LIN {X 0,Y 274.208,Z 1013.96,A -85,B 0,C 180,E1 12726.209,E2 12726.209} C_VEL
LIN {X 0,Y 266.688,Z 1024.123,A -85,B 0,C 180,E1 12721.914,E2 12721.914} C_VEL
LIN {X 0,Y 259.994,Z 1033.612,A -85,B 0,C 180,E1 12716.988,E2 12716.988} C_VEL
LIN {X 0,Y 254.913,Z 1041.187,A -85,B 0,C 180,E1 12711.878,E2 12711.878} C_VEL
LIN {X 0,Y 251.523,Z 1047.053,A -85,B 0,C 180,E1 12706.87,E2 12706.87} C_VEL
LIN {X 0,Y 249.285,Z 1051.783,A -85,B 0,C 180,E1 12701.335,E2 12701.335} C_VEL
LIN {X 0,Y 248.38,Z 1054.512,A -85,B 0,C 180,E1 12696.704,E2 12696.704} C_VEL
LIN {X 0,Y 248.075,Z 1056.133,A -85,B 0,C 180,E1 12692.31,E2 12692.31} C_VEL
LIN {X 0,Y 248.004,Z 1056.84,A -85,B 0,C 180,E1 12687.689,E2 12687.689} C_VEL
LIN {X 0,Y 248.137,Z 1056.355,A -85,B 0,C 180,E1 12682.591,E2 12682.591} C_VEL
LIN {X 0,Y 248.642,Z 1054.659,A -85,B 0,C 180,E1 12677.694,E2 12677.694} C_VEL
LIN {X 0,Y 249.87,Z 1051.971,A -85,B 0,C 180,E1 12673.015,E2 12673.015} C_VEL
LIN {X 0,Y 252.833,Z 1046.979,A -85,B 0,C 180,E1 12667.141,E2 12667.141} C_VEL
LIN {X 0,Y 256.876,Z 1041.112,A -85,B 0,C 180,E1 12662.154,E2 12662.154} C_VEL
LIN {X 0,Y 263.072,Z 1033.015,A -85,B 0,C 180,E1 12656.817,E2 12656.817} C_VEL
LIN {X 0,Y 270.365,Z 1023.771,A -85,B 0,C 180,E1 12652.127,E2 12652.127} C_VEL
LIN {X 0,Y 279.2,Z 1012.904,A -85,B 0,C 180,E1 12647.679,E2 12647.679} C_VEL
LIN {X 0,Y 288.948,Z 1000.521,A -85,B 0,C 180,E1 12643.678,E2 12643.678} C_VEL
LIN {X 0,Y 299.389,Z 987.042,A -85,B 0,C 180,E1 12640.11,E2 12640.11} C_VEL
LIN {X 0,Y 310.24,Z 972.088,A -85,B 0,C 180,E1 12636.937,E2 12636.937} C_VEL
LIN {X 0,Y 320.673,Z 956.975,A -85,B 0,C 180,E1 12634.28,E2 12634.28} C_VEL
LIN {X 0,Y 332.382,Z 938.579,A -85,B 0,C 180,E1 12631.643,E2 12631.643} C_VEL
LIN {X 0,Y 341.93,Z 922.312,A -85,B 0,C 180,E1 12629.715,E2 12629.715} C_VEL
LIN {X 0,Y 353.262,Z 901.024,A -85,B 0,C 180,E1 12627.634,E2 12627.634} C_VEL
LIN {X 0,Y 362.036,Z 882.572,A -85,B 0,C 180,E1 12626.155,E2 12626.155} C_VEL
LIN {X 0,Y 371.461,Z 860.323,A -85,B 0,C 180,E1 12624.686,E2 12624.686} C_VEL
LIN {X 0,Y 379.053,Z 839.359,A -85,B 0,C 180,E1 12623.558,E2 12623.558} C_VEL
LIN {X 0,Y 386.253,Z 816.382,A -85,B 0,C 180,E1 12622.555,E2 12622.555} C_VEL
LIN {X 0,Y 392.125,Z 792.972,A -85,B 0,C 180,E1 12621.762,E2 12621.762} C_VEL
LIN {X 0,Y 396.905,Z 769.324,A -85,B 0,C 180,E1 12621.142,E2 12621.142} C_VEL
LIN {X 0,Y 400.292,Z 744.689,A -85,B 0,C 180,E1 12620.665,E2 12620.665} C_VEL
LIN {X 0,Y 415.264,Z 580.278,A -85,B 0,C 180,E1 12618.096,E2 12618.096} C_VEL
LIN {X 0,Y 415.202,Z 577.101,A -85,B 0,C 180,E1 12617.904,E2 12617.904} C_VEL
LIN {X 0,Y 414.493,Z 574.251,A -85,B 0,C 180,E1 12617.461,E2 12617.461} C_VEL
LIN {X 0,Y 412.986,Z 571.866,A -85,B 0,C 180,E1 12616.684,E2 12616.684} C_VEL
LIN {X 0,Y 410.26,Z 568.824,A -85,B 0,C 180,E1 12615.251,E2 12615.251} C_VEL
LIN {X 0,Y 405.888,Z 561,A -85,B 0,C 180,E1 12612.376,E2 12612.376} C_VEL
LIN {X 0,Y 403.184,Z 556.35,A -85,B 0,C 180,E1 12610.214,E2 12610.214} C_VEL
LIN {X 0,Y 401.232,Z 552.898,A -85,B 0,C 180,E1 12608.311,E2 12608.311} C_VEL
LIN {X 0,Y 399.029,Z 548.877,A -85,B 0,C 180,E1 12605.464,E2 12605.464} C_VEL
LIN {X 0,Y 397.148,Z 544.545,A -85,B 0,C 180,E1 12599.134,E2 12599.134} C_VEL
LIN {X 0,Y 399.305,Z 549.372,A -85,B 0,C 180,E1 12592.446,E2 12592.446} C_VEL
LIN {X 0,Y 402.053,Z 554.34,A -85,B 0,C 180,E1 12589.178,E2 12589.178} C_VEL
LIN {X 0,Y 404.963,Z 559.417,A -85,B 0,C 180,E1 12586.652,E2 12586.652} C_VEL
LIN {X 0,Y 408.355,Z 565.354,A -85,B 0,C 180,E1 12584.265,E2 12584.265} C_VEL
LIN {X 0,Y 413.221,Z 576.035,A -85,B 0,C 180,E1 12581.314,E2 12581.314} C_VEL
LIN {X 0,Y 396.472,Z 755.864,A -85,B 0,C 180,E1 12578.511,E2 12578.511} C_VEL
LIN {X 0,Y 392.307,Z 782.562,A -85,B 0,C 180,E1 12577.987,E2 12577.987} C_VEL
LIN {X 0,Y 387.69,Z 803.875,A -85,B 0,C 180,E1 12577.456,E2 12577.456} C_VEL
LIN {X 0,Y 381.104,Z 828.129,A -85,B 0,C 180,E1 12576.676,E2 12576.676} C_VEL
LIN {X 0,Y 374.28,Z 848.813,A -85,B 0,C 180,E1 12575.828,E2 12575.828} C_VEL
LIN {X 0,Y 365.745,Z 871.344,A -85,B 0,C 180,E1 12574.679,E2 12574.679} C_VEL
LIN {X 0,Y 356.44,Z 892.358,A -85,B 0,C 180,E1 12573.331,E2 12573.331} C_VEL
LIN {X 0,Y 346.382,Z 912.781,A -85,B 0,C 180,E1 12571.744,E2 12571.744} C_VEL
LIN {X 0,Y 335.391,Z 932.564,A -85,B 0,C 180,E1 12569.833,E2 12569.833} C_VEL
LIN {X 0,Y 324.92,Z 949.901,A -85,B 0,C 180,E1 12567.808,E2 12567.808} C_VEL
LIN {X 0,Y 312.929,Z 968.085,A -85,B 0,C 180,E1 12565.203,E2 12565.203} C_VEL
LIN {X 0,Y 302.254,Z 983.196,A -85,B 0,C 180,E1 12562.556,E2 12562.556} C_VEL
LIN {X 0,Y 290.029,Z 999.531,A -85,B 0,C 180,E1 12559.027,E2 12559.027} C_VEL
LIN {X 0,Y 279.971,Z 1012.354,A -85,B 0,C 180,E1 12555.584,E2 12555.584} C_VEL
LIN {X 0,Y 269.185,Z 1025.802,A -85,B 0,C 180,E1 12551.107,E2 12551.107} C_VEL
LIN {X 0,Y 260.773,Z 1036.213,A -85,B 0,C 180,E1 12546.738,E2 12546.738} C_VEL
LIN {X 0,Y 252.94,Z 1046.262,A -85,B 0,C 180,E1 12541.454,E2 12541.454} C_VEL
LIN {X 0,Y 247.478,Z 1053.723,A -85,B 0,C 180,E1 12536.387,E2 12536.387} C_VEL
LIN {X 0,Y 243.363,Z 1060.291,A -85,B 0,C 180,E1 12530.692,E2 12530.692} C_VEL
LIN {X 0,Y 241.068,Z 1064.832,A -85,B 0,C 180,E1 12525.148,E2 12525.148} C_VEL
LIN {X 0,Y 240.171,Z 1067.628,A -85,B 0,C 180,E1 12520.313,E2 12520.313} C_VEL
LIN {X 0,Y 239.975,Z 1069.472,A -85,B 0,C 180,E1 12515.02,E2 12515.02} C_VEL
LIN {X 0,Y 240.024,Z 1069.836,A -85,B 0,C 180,E1 12510,E2 12510} C_VEL
LIN {X 0,Y 239.982,Z 1069.112,A -85,B 0,C 180,E1 12505.46,E2 12505.46} C_VEL
LIN {X 0,Y 240.062,Z 1067.493,A -85,B 0,C 180,E1 12501.135,E2 12501.135} C_VEL
LIN {X 0,Y 240.688,Z 1064.623,A -85,B 0,C 180,E1 12496.303,E2 12496.303} C_VEL
LIN {X 0,Y 242.774,Z 1059.401,A -85,B 0,C 180,E1 12490.262,E2 12490.262} C_VEL
LIN {X 0,Y 245.938,Z 1053.504,A -85,B 0,C 180,E1 12485.244,E2 12485.244} C_VEL
LIN {X 0,Y 251.056,Z 1045.569,A -85,B 0,C 180,E1 12479.879,E2 12479.879} C_VEL
LIN {X 0,Y 257.954,Z 1035.663,A -85,B 0,C 180,E1 12474.721,E2 12474.721} C_VEL
LIN {X 0,Y 266.254,Z 1024.474,A -85,B 0,C 180,E1 12470.006,E2 12470.006} C_VEL
LIN {X 0,Y 275.494,Z 1011.927,A -85,B 0,C 180,E1 12465.825,E2 12465.825} C_VEL
LIN {X 0,Y 285.04,Z 998.91,A -85,B 0,C 180,E1 12462.255,E2 12462.255} C_VEL
LIN {X 0,Y 296.15,Z 983.09,A -85,B 0,C 180,E1 12458.747,E2 12458.747} C_VEL
LIN {X 0,Y 306.358,Z 967.847,A -85,B 0,C 180,E1 12455.979,E2 12455.979} C_VEL
LIN {X 0,Y 317.965,Z 949.305,A -85,B 0,C 180,E1 12453.23,E2 12453.23} C_VEL
LIN {X 0,Y 327.782,Z 932.315,A -85,B 0,C 180,E1 12451.168,E2 12451.168} C_VEL
LIN {X 0,Y 338.722,Z 911.666,A -85,B 0,C 180,E1 12449.1,E2 12449.1} C_VEL
LIN {X 0,Y 347.872,Z 892.386,A -85,B 0,C 180,E1 12447.536,E2 12447.536} C_VEL
LIN {X 0,Y 357.142,Z 870.654,A -85,B 0,C 180,E1 12446.076,E2 12446.076} C_VEL
LIN {X 0,Y 364.973,Z 849.253,A -85,B 0,C 180,E1 12444.931,E2 12444.931} C_VEL
LIN {X 0,Y 371.657,Z 828.377,A -85,B 0,C 180,E1 12444.024,E2 12444.024} C_VEL
LIN {X 0,Y 378.109,Z 803.884,A -85,B 0,C 180,E1 12443.192,E2 12443.192} C_VEL
LIN {X 0,Y 382.633,Z 782.361,A -85,B 0,C 180,E1 12442.628,E2 12442.628} C_VEL
LIN {X 0,Y 386.671,Z 755.374,A -85,B 0,C 180,E1 12442.077,E2 12442.077} C_VEL
LIN {X 0,Y 403.402,Z 568.894,A -85,B 0,C 180,E1 12439.098,E2 12439.098} C_VEL
LIN {X 0,Y 398.244,Z 557.633,A -85,B 0,C 180,E1 12436.332,E2 12436.332} C_VEL
LIN {X 0,Y 393.971,Z 550.114,A -85,B 0,C 180,E1 12433.727,E2 12433.727} C_VEL
LIN {X 0,Y 390.379,Z 543.824,A -85,B 0,C 180,E1 12431.075,E2 12431.075} C_VEL
LIN {X 0,Y 387.521,Z 539.169,A -85,B 0,C 180,E1 12428.457,E2 12428.457} C_VEL
LIN {X 0,Y 385.179,Z 535.036,A -85,B 0,C 180,E1 12425.512,E2 12425.512} C_VEL
LIN {X 0,Y 383.121,Z 530.299,A -85,B 0,C 180,E1 12418.654,E2 12418.654} C_VEL
LIN {X 0,Y 385.47,Z 535.482,A -85,B 0,C 180,E1 12411.648,E2 12411.648} C_VEL
LIN {X 0,Y 388.46,Z 540.683,A -85,B 0,C 180,E1 12408.192,E2 12408.192} C_VEL
LIN {X 0,Y 391.35,Z 545.617,A -85,B 0,C 180,E1 12405.726,E2 12405.726} C_VEL
LIN {X 0,Y 395.237,Z 552.118,A -85,B 0,C 180,E1 12403.048,E2 12403.048} C_VEL
LIN {X 0,Y 400.428,Z 561.515,A -85,B 0,C 180,E1 12400.071,E2 12400.071} C_VEL
LIN {X 0,Y 403.438,Z 567.456,A -85,B 0,C 180,E1 12398.544,E2 12398.544} C_VEL
LIN {X 0,Y 387.142,Z 748.135,A -85,B 0,C 180,E1 12395.669,E2 12395.669} C_VEL
LIN {X 0,Y 383.184,Z 774.56,A -85,B 0,C 180,E1 12395.108,E2 12395.108} C_VEL
LIN {X 0,Y 378.931,Z 795.289,A -85,B 0,C 180,E1 12394.524,E2 12394.524} C_VEL
LIN {X 0,Y 372.699,Z 819.594,A -85,B 0,C 180,E1 12393.646,E2 12393.646} C_VEL
LIN {X 0,Y 366.228,Z 840.253,A -85,B 0,C 180,E1 12392.698,E2 12392.698} C_VEL
LIN {X 0,Y 358.451,Z 861.898,A -85,B 0,C 180,E1 12391.484,E2 12391.484} C_VEL
LIN {X 0,Y 349.307,Z 883.51,A -85,B 0,C 180,E1 12389.986,E2 12389.986} C_VEL
LIN {X 0,Y 340.037,Z 903.213,A -85,B 0,C 180,E1 12388.33,E2 12388.33} C_VEL
LIN {X 0,Y 329.424,Z 923.215,A -85,B 0,C 180,E1 12386.27,E2 12386.27} C_VEL
LIN {X 0,Y 319.951,Z 939.603,A -85,B 0,C 180,E1 12384.239,E2 12384.239} C_VEL
LIN {X 0,Y 308.213,Z 958.246,A -85,B 0,C 180,E1 12381.429,E2 12381.429} C_VEL
LIN {X 0,Y 298.169,Z 973.091,A -85,B 0,C 180,E1 12378.692,E2 12378.692} C_VEL
LIN {X 0,Y 286.701,Z 989.113,A -85,B 0,C 180,E1 12375.07,E2 12375.07} C_VEL
LIN {X 0,Y 277.303,Z 1001.648,A -85,B 0,C 180,E1 12371.564,E2 12371.564} C_VEL
LIN {X 0,Y 267.668,Z 1014.257,A -85,B 0,C 180,E1 12367.24,E2 12367.24} C_VEL
LIN {X 0,Y 259.797,Z 1024.412,A -85,B 0,C 180,E1 12362.866,E2 12362.866} C_VEL
LIN {X 0,Y 252.758,Z 1033.885,A -85,B 0,C 180,E1 12357.827,E2 12357.827} C_VEL
LIN {X 0,Y 247.387,Z 1041.451,A -85,B 0,C 180,E1 12352.58,E2 12352.58} C_VEL
LIN {X 0,Y 243.652,Z 1047.556,A -85,B 0,C 180,E1 12347.186,E2 12347.186} C_VEL
LIN {X 0,Y 241.317,Z 1052.178,A -85,B 0,C 180,E1 12341.472,E2 12341.472} C_VEL
LIN {X 0,Y 240.381,Z 1054.854,A -85,B 0,C 180,E1 12336.688,E2 12336.688} C_VEL
LIN {X 0,Y 240.066,Z 1056.49,A -85,B 0,C 180,E1 12331.909,E2 12331.909} C_VEL
LIN {X 0,Y 240.014,Z 1057.097,A -85,B 0,C 180,E1 12326.895,E2 12326.895} C_VEL
LIN {X 0,Y 240.171,Z 1056.429,A -85,B 0,C 180,E1 12321.862,E2 12321.862} C_VEL
LIN {X 0,Y 240.764,Z 1054.748,A -85,B 0,C 180,E1 12317.041,E2 12317.041} C_VEL
LIN {X 0,Y 242.354,Z 1051.699,A -85,B 0,C 180,E1 12311.726,E2 12311.726} C_VEL
LIN {X 0,Y 245.555,Z 1046.718,A -85,B 0,C 180,E1 12305.971,E2 12305.971} C_VEL
LIN {X 0,Y 249.825,Z 1040.987,A -85,B 0,C 180,E1 12301.034,E2 12301.034} C_VEL
LIN {X 0,Y 256.801,Z 1032.373,A -85,B 0,C 180,E1 12295.356,E2 12295.356} C_VEL
LIN {X 0,Y 264.258,Z 1023.467,A -85,B 0,C 180,E1 12290.81,E2 12290.81} C_VEL
LIN {X 0,Y 274.029,Z 1011.899,A -85,B 0,C 180,E1 12286.11,E2 12286.11} C_VEL
LIN {X 0,Y 283.806,Z 1000.013,A -85,B 0,C 180,E1 12282.281,E2 12282.281} C_VEL
LIN {X 0,Y 295.269,Z 985.638,A -85,B 0,C 180,E1 12278.533,E2 12278.533} C_VEL
LIN {X 0,Y 305.967,Z 971.336,A -85,B 0,C 180,E1 12275.539,E2 12275.539} C_VEL
LIN {X 0,Y 317.421,Z 955.203,A -85,B 0,C 180,E1 12272.748,E2 12272.748} C_VEL
LIN {X 0,Y 328.836,Z 937.519,A -85,B 0,C 180,E1 12270.281,E2 12270.281} C_VEL
LIN {X 0,Y 339.38,Z 919.914,A -85,B 0,C 180,E1 12268.246,E2 12268.246} C_VEL
LIN {X 0,Y 350.287,Z 899.549,A -85,B 0,C 180,E1 12266.323,E2 12266.323} C_VEL
LIN {X 0,Y 358.905,Z 881.731,A -85,B 0,C 180,E1 12264.93,E2 12264.93} C_VEL
LIN {X 0,Y 368.941,Z 858.156,A -85,B 0,C 180,E1 12263.42,E2 12263.42} C_VEL
LIN {X 0,Y 376.287,Z 838.102,A -85,B 0,C 180,E1 12262.373,E2 12262.373} C_VEL
LIN {X 0,Y 383.819,Z 813.925,A -85,B 0,C 180,E1 12261.358,E2 12261.358} C_VEL
LIN {X 0,Y 389.378,Z 791.903,A -85,B 0,C 180,E1 12260.635,E2 12260.635} C_VEL
LIN {X 0,Y 394.305,Z 767.229,A -85,B 0,C 180,E1 12260.014,E2 12260.014} C_VEL
LIN {X 0,Y 397.509,Z 743.917,A -85,B 0,C 180,E1 12259.577,E2 12259.577} C_VEL
LIN {X 0,Y 413.233,Z 574.497,A -85,B 0,C 180,E1 12256.939,E2 12256.939} C_VEL
LIN {X 0,Y 410.26,Z 568.824,A -85,B 0,C 180,E1 12255.251,E2 12255.251} C_VEL
LIN {X 0,Y 408.323,Z 566.877,A -85,B 0,C 180,E1 12254.153,E2 12254.153} C_VEL
LIN {X 0,Y 402.936,Z 565.423,A -85,B 0,C 180,E1 12250.841,E2 12250.841} C_VEL
LIN {X 0,Y 402.359,Z 564.773,A -85,B 0,C 180,E1 12250.379,E2 12250.379} C_VEL
LIN {X 0,Y 399.981,Z 560.605,A -85,B 0,C 180,E1 12248.047,E2 12248.047} C_VEL
LIN {X 0,Y 397.86,Z 556.677,A -85,B 0,C 180,E1 12245.191,E2 12245.191} C_VEL
LIN {X 0,Y 396.169,Z 552.519,A -85,B 0,C 180,E1 12239.132,E2 12239.132} C_VEL
LIN {X 0,Y 398.223,Z 557.306,A -85,B 0,C 180,E1 12232.57,E2 12232.57} C_VEL
LIN {X 0,Y 400.781,Z 562.036,A -85,B 0,C 180,E1 12229.434,E2 12229.434} C_VEL
LIN {X 0,Y 403.525,Z 566.964,A -85,B 0,C 180,E1 12226.968,E2 12226.968} C_VEL
LIN {X 0,Y 406.77,Z 572.828,A -85,B 0,C 180,E1 12224.605,E2 12224.605} C_VEL
LIN {X 0,Y 410.341,Z 581.211,A -85,B 0,C 180,E1 12222.297,E2 12222.297} C_VEL
LIN {X 0,Y 393.726,Z 755.676,A -85,B 0,C 180,E1 12219.606,E2 12219.606} C_VEL
LIN {X 0,Y 389.508,Z 782.287,A -85,B 0,C 180,E1 12219.091,E2 12219.091} C_VEL
LIN {X 0,Y 384.811,Z 803.636,A -85,B 0,C 180,E1 12218.571,E2 12218.571} C_VEL
LIN {X 0,Y 377.998,Z 828.265,A -85,B 0,C 180,E1 12217.794,E2 12217.794} C_VEL
LIN {X 0,Y 371.058,Z 848.906,A -85,B 0,C 180,E1 12216.961,E2 12216.961} C_VEL
LIN {X 0,Y 362.252,Z 871.633,A -85,B 0,C 180,E1 12215.818,E2 12215.818} C_VEL
LIN {X 0,Y 352.801,Z 892.535,A -85,B 0,C 180,E1 12214.493,E2 12214.493} C_VEL
LIN {X 0,Y 342.316,Z 913.337,A -85,B 0,C 180,E1 12212.892,E2 12212.892} C_VEL
LIN {X 0,Y 331.006,Z 933.122,A -85,B 0,C 180,E1 12210.987,E2 12210.987} C_VEL
LIN {X 0,Y 319.94,Z 950.948,A -85,B 0,C 180,E1 12208.905,E2 12208.905} C_VEL
LIN {X 0,Y 307.654,Z 968.923,A -85,B 0,C 180,E1 12206.306,E2 12206.306} C_VEL
LIN {X 0,Y 296.416,Z 984.325,A -85,B 0,C 180,E1 12203.58,E2 12203.58} C_VEL
LIN {X 0,Y 284.108,Z 1000.112,A -85,B 0,C 180,E1 12200.106,E2 12200.106} C_VEL
LIN {X 0,Y 274.242,Z 1012.221,A -85,B 0,C 180,E1 12196.82,E2 12196.82} C_VEL
LIN {X 0,Y 262.999,Z 1025.652,A -85,B 0,C 180,E1 12192.294,E2 12192.294} C_VEL
LIN {X 0,Y 254.566,Z 1035.589,A -85,B 0,C 180,E1 12188.073,E2 12188.073} C_VEL
LIN {X 0,Y 246.508,Z 1045.405,A -85,B 0,C 180,E1 12182.898,E2 12182.898} C_VEL
LIN {X 0,Y 240.341,Z 1053.235,A -85,B 0,C 180,E1 12177.503,E2 12177.503} C_VEL
LIN {X 0,Y 235.845,Z 1059.872,A -85,B 0,C 180,E1 12171.645,E2 12171.645} C_VEL
LIN {X 0,Y 233.202,Z 1064.635,A -85,B 0,C 180,E1 12165.672,E2 12165.672} C_VEL
LIN {X 0,Y 232.206,Z 1067.427,A -85,B 0,C 180,E1 12160.67,E2 12160.67} C_VEL
LIN {X 0,Y 231.976,Z 1069.266,A -85,B 0,C 180,E1 12155.193,E2 12155.193} C_VEL
LIN {X 0,Y 232.019,Z 1069.641,A -85,B 0,C 180,E1 12150.247,E2 12150.247} C_VEL
LIN {X 0,Y 231.984,Z 1068.958,A -85,B 0,C 180,E1 12145.55,E2 12145.55} C_VEL
LIN {X 0,Y 232.065,Z 1067.379,A -85,B 0,C 180,E1 12141.077,E2 12141.077} C_VEL
LIN {X 0,Y 232.701,Z 1064.624,A -85,B 0,C 180,E1 12136.192,E2 12136.192} C_VEL
LIN {X 0,Y 234.7,Z 1059.909,A -85,B 0,C 180,E1 12130.31,E2 12130.31} C_VEL
LIN {X 0,Y 238.268,Z 1053.553,A -85,B 0,C 180,E1 12124.657,E2 12124.657} C_VEL
LIN {X 0,Y 243.373,Z 1046.025,A -85,B 0,C 180,E1 12119.373,E2 12119.373} C_VEL
LIN {X 0,Y 250.514,Z 1036.315,A -85,B 0,C 180,E1 12114.075,E2 12114.075} C_VEL
LIN {X 0,Y 258.183,Z 1026.358,A -85,B 0,C 180,E1 12109.703,E2 12109.703} C_VEL
LIN {X 0,Y 268.617,Z 1012.911,A -85,B 0,C 180,E1 12104.989,E2 12104.989} C_VEL
LIN {X 0,Y 277.893,Z 1000.729,A -85,B 0,C 180,E1 12101.547,E2 12101.547} C_VEL
LIN {X 0,Y 289.353,Z 985.184,A -85,B 0,C 180,E1 12097.959,E2 12097.959} C_VEL
LIN {X 0,Y 299.7,Z 970.261,A -85,B 0,C 180,E1 12095.175,E2 12095.175} C_VEL
LIN {X 0,Y 311.165,Z 952.835,A -85,B 0,C 180,E1 12092.487,E2 12092.487} C_VEL
LIN {X 0,Y 322.546,Z 933.775,A -85,B 0,C 180,E1 12090.129,E2 12090.129} C_VEL
LIN {X 0,Y 333.349,Z 914.165,A -85,B 0,C 180,E1 12088.132,E2 12088.132} C_VEL
LIN {X 0,Y 343.386,Z 893.65,A -85,B 0,C 180,E1 12086.456,E2 12086.456} C_VEL
LIN {X 0,Y 352.222,Z 873.559,A -85,B 0,C 180,E1 12085.099,E2 12085.099} C_VEL
LIN {X 0,Y 360.979,Z 850.598,A -85,B 0,C 180,E1 12083.854,E2 12083.854} C_VEL
LIN {X 0,Y 367.441,Z 830.993,A -85,B 0,C 180,E1 12083,E2 12083} C_VEL
LIN {X 0,Y 374.212,Z 806.578,A -85,B 0,C 180,E1 12082.153,E2 12082.153} C_VEL
LIN {X 0,Y 379.062,Z 784.332,A -85,B 0,C 180,E1 12081.567,E2 12081.567} C_VEL
LIN {X 0,Y 383.117,Z 759.514,A -85,B 0,C 180,E1 12081.049,E2 12081.049} C_VEL
LIN {X 0,Y 388.393,Z 704.087,A -85,B 0,C 180,E1 12080.146,E2 12080.146} C_VEL
LIN {X 0,Y 400.252,Z 573.446,A -85,B 0,C 180,E1 12078.083,E2 12078.083} C_VEL
LIN {X 0,Y 395.946,Z 563.972,A -85,B 0,C 180,E1 12075.639,E2 12075.639} C_VEL
LIN {X 0,Y 391.725,Z 556.337,A -85,B 0,C 180,E1 12072.906,E2 12072.906} C_VEL
LIN {X 0,Y 388.594,Z 550.898,A -85,B 0,C 180,E1 12070.452,E2 12070.452} C_VEL
LIN {X 0,Y 386.254,Z 546.876,A -85,B 0,C 180,E1 12068.185,E2 12068.185} C_VEL
LIN {X 0,Y 383.997,Z 542.829,A -85,B 0,C 180,E1 12065.229,E2 12065.229} C_VEL
LIN {X 0,Y 382.142,Z 538.278,A -85,B 0,C 180,E1 12058.651,E2 12058.651} C_VEL
LIN {X 0,Y 384.382,Z 543.419,A -85,B 0,C 180,E1 12051.774,E2 12051.774} C_VEL
LIN {X 0,Y 387.171,Z 548.383,A -85,B 0,C 180,E1 12048.454,E2 12048.454} C_VEL
LIN {X 0,Y 389.894,Z 553.166,A -85,B 0,C 180,E1 12046.051,E2 12046.051} C_VEL
LIN {X 0,Y 393.621,Z 559.599,A -85,B 0,C 180,E1 12043.395,E2 12043.395} C_VEL
LIN {X 0,Y 398.687,Z 569.021,A -85,B 0,C 180,E1 12040.401,E2 12040.401} C_VEL
LIN {X 0,Y 400.284,Z 572.367,A -85,B 0,C 180,E1 12039.544,E2 12039.544} C_VEL
LIN {X 0,Y 384.057,Z 748.302,A -85,B 0,C 180,E1 12036.767,E2 12036.767} C_VEL
LIN {X 0,Y 380.026,Z 774.745,A -85,B 0,C 180,E1 12036.213,E2 12036.213} C_VEL
LIN {X 0,Y 375.691,Z 795.491,A -85,B 0,C 180,E1 12035.638,E2 12035.638} C_VEL
LIN {X 0,Y 369.224,Z 820.189,A -85,B 0,C 180,E1 12034.756,E2 12034.756} C_VEL
LIN {X 0,Y 362.643,Z 840.766,A -85,B 0,C 180,E1 12033.822,E2 12033.822} C_VEL
LIN {X 0,Y 354.698,Z 862.408,A -85,B 0,C 180,E1 12032.621,E2 12032.621} C_VEL
LIN {X 0,Y 345.362,Z 883.966,A -85,B 0,C 180,E1 12031.139,E2 12031.139} C_VEL
LIN {X 0,Y 335.768,Z 903.879,A -85,B 0,C 180,E1 12029.477,E2 12029.477} C_VEL
LIN {X 0,Y 325.015,Z 923.613,A -85,B 0,C 180,E1 12027.452,E2 12027.452} C_VEL
LIN {X 0,Y 314.859,Z 940.708,A -85,B 0,C 180,E1 12025.336,E2 12025.336} C_VEL
LIN {X 0,Y 303.227,Z 958.602,A -85,B 0,C 180,E1 12022.627,E2 12022.627} C_VEL
LIN {X 0,Y 292.874,Z 973.436,A -85,B 0,C 180,E1 12019.885,E2 12019.885} C_VEL
LIN {X 0,Y 281.008,Z 989.437,A -85,B 0,C 180,E1 12016.246,E2 12016.246} C_VEL
LIN {X 0,Y 271.257,Z 1001.963,A -85,B 0,C 180,E1 12012.707,E2 12012.707} C_VEL
LIN {X 0,Y 261.14,Z 1014.647,A -85,B 0,C 180,E1 12008.285,E2 12008.285} C_VEL
LIN {X 0,Y 252.983,Z 1024.7,A -85,B 0,C 180,E1 12003.868,E2 12003.868} C_VEL
LIN {X 0,Y 245.579,Z 1034.158,A -85,B 0,C 180,E1 11998.714,E2 11998.714} C_VEL
LIN {X 0,Y 239.901,Z 1041.714,A -85,B 0,C 180,E1 11993.325,E2 11993.325} C_VEL
LIN {X 0,Y 235.924,Z 1047.812,A -85,B 0,C 180,E1 11987.767,E2 11987.767} C_VEL
LIN {X 0,Y 233.421,Z 1052.417,A -85,B 0,C 180,E1 11981.865,E2 11981.865} C_VEL
LIN {X 0,Y 232.411,Z 1055.085,A -85,B 0,C 180,E1 11976.919,E2 11976.919} C_VEL
LIN {X 0,Y 232.071,Z 1056.714,A -85,B 0,C 180,E1 11971.975,E2 11971.975} C_VEL
LIN {X 0,Y 232.018,Z 1057.307,A -85,B 0,C 180,E1 11966.788,E2 11966.788} C_VEL
LIN {X 0,Y 232.196,Z 1056.634,A -85,B 0,C 180,E1 11961.581,E2 11961.581} C_VEL
LIN {X 0,Y 232.853,Z 1054.948,A -85,B 0,C 180,E1 11956.592,E2 11956.592} C_VEL
LIN {X 0,Y 234.592,Z 1051.893,A -85,B 0,C 180,E1 11951.099,E2 11951.099} C_VEL
LIN {X 0,Y 238.088,Z 1046.847,A -85,B 0,C 180,E1 11945.112,E2 11945.112} C_VEL
LIN {X 0,Y 242.615,Z 1041.161,A -85,B 0,C 180,E1 11940.087,E2 11940.087} C_VEL
LIN {X 0,Y 250.02,Z 1032.531,A -85,B 0,C 180,E1 11934.275,E2 11934.275} C_VEL
LIN {X 0,Y 257.882,Z 1023.616,A -85,B 0,C 180,E1 11929.646,E2 11929.646} C_VEL
LIN {X 0,Y 268.413,Z 1011.672,A -85,B 0,C 180,E1 11924.754,E2 11924.754} C_VEL
LIN {X 0,Y 278.302,Z 1000.135,A -85,B 0,C 180,E1 11921.019,E2 11921.019} C_VEL
LIN {X 0,Y 290.19,Z 985.74,A -85,B 0,C 180,E1 11917.256,E2 11917.256} C_VEL
LIN {X 0,Y 301.246,Z 971.426,A -85,B 0,C 180,E1 11914.261,E2 11914.261} C_VEL
LIN {X 0,Y 313.044,Z 955.275,A -85,B 0,C 180,E1 11911.48,E2 11911.48} C_VEL
LIN {X 0,Y 324.773,Z 937.569,A -85,B 0,C 180,E1 11909.031,E2 11909.031} C_VEL
LIN {X 0,Y 335.952,Z 919.34,A -85,B 0,C 180,E1 11906.951,E2 11906.951} C_VEL
LIN {X 0,Y 346.746,Z 899.544,A -85,B 0,C 180,E1 11905.114,E2 11905.114} C_VEL
LIN {X 0,Y 355.593,Z 881.622,A -85,B 0,C 180,E1 11903.736,E2 11903.736} C_VEL
LIN {X 0,Y 365.537,Z 858.721,A -85,B 0,C 180,E1 11902.29,E2 11902.29} C_VEL
LIN {X 0,Y 372.878,Z 839.111,A -85,B 0,C 180,E1 11901.277,E2 11901.277} C_VEL
LIN {X 0,Y 380.332,Z 815.968,A -85,B 0,C 180,E1 11900.306,E2 11900.306} C_VEL
LIN {X 0,Y 386.25,Z 793.125,A -85,B 0,C 180,E1 11899.56,E2 11899.56} C_VEL
LIN {X 0,Y 391.244,Z 769.089,A -85,B 0,C 180,E1 11898.954,E2 11898.954} C_VEL
LIN {X 0,Y 394.683,Z 744.791,A -85,B 0,C 180,E1 11898.5,E2 11898.5} C_VEL
LIN {X 0,Y 410.348,Z 579.625,A -85,B 0,C 180,E1 11895.946,E2 11895.946} C_VEL
LIN {X 0,Y 405.942,Z 571.377,A -85,B 0,C 180,E1 11893.17,E2 11893.17} C_VEL
LIN {X 0,Y 402.359,Z 564.773,A -85,B 0,C 180,E1 11890.379,E2 11890.379} C_VEL
LIN {X 0,Y 400.956,Z 563.777,A -85,B 0,C 180,E1 11889.221,E2 11889.221} C_VEL
LIN {X 0,Y 397.256,Z 564.937,A -85,B 0,C 180,E1 11885.734,E2 11885.734} C_VEL
LIN {X 0,Y 396.971,Z 564.739,A -85,B 0,C 180,E1 11885.334,E2 11885.334} C_VEL
LIN {X 0,Y 395.189,Z 560.495,A -85,B 0,C 180,E1 11879.13,E2 11879.13} C_VEL
LIN {X 0,Y 397.102,Z 565.119,A -85,B 0,C 180,E1 11872.767,E2 11872.767} C_VEL
LIN {X 0,Y 399.583,Z 569.876,A -85,B 0,C 180,E1 11869.62,E2 11869.62} C_VEL
LIN {X 0,Y 402.269,Z 574.828,A -85,B 0,C 180,E1 11867.146,E2 11867.146} C_VEL
LIN {X 0,Y 405.294,Z 580.545,A -85,B 0,C 180,E1 11864.877,E2 11864.877} C_VEL
LIN {X 0,Y 407.597,Z 586.184,A -85,B 0,C 180,E1 11863.301,E2 11863.301} C_VEL
LIN {X 0,Y 391.12,Z 755.536,A -85,B 0,C 180,E1 11860.715,E2 11860.715} C_VEL
LIN {X 0,Y 386.856,Z 782.013,A -85,B 0,C 180,E1 11860.211,E2 11860.211} C_VEL
LIN {X 0,Y 382.072,Z 803.435,A -85,B 0,C 180,E1 11859.701,E2 11859.701} C_VEL
LIN {X 0,Y 375.038,Z 828.403,A -85,B 0,C 180,E1 11858.929,E2 11858.929} C_VEL
LIN {X 0,Y 367.984,Z 849.001,A -85,B 0,C 180,E1 11858.114,E2 11858.114} C_VEL
LIN {X 0,Y 359.022,Z 871.665,A -85,B 0,C 180,E1 11856.993,E2 11856.993} C_VEL
LIN {X 0,Y 349.433,Z 892.46,A -85,B 0,C 180,E1 11855.696,E2 11855.696} C_VEL
LIN {X 0,Y 338.891,Z 912.953,A -85,B 0,C 180,E1 11854.144,E2 11854.144} C_VEL
LIN {X 0,Y 327.505,Z 932.463,A -85,B 0,C 180,E1 11852.299,E2 11852.299} C_VEL
LIN {X 0,Y 316.516,Z 949.77,A -85,B 0,C 180,E1 11850.313,E2 11850.313} C_VEL
LIN {X 0,Y 303.867,Z 967.902,A -85,B 0,C 180,E1 11847.744,E2 11847.744} C_VEL
LIN {X 0,Y 293.193,Z 982.14,A -85,B 0,C 180,E1 11845.275,E2 11845.275} C_VEL
LIN {X 0,Y 280.683,Z 997.872,A -85,B 0,C 180,E1 11841.932,E2 11841.932} C_VEL
LIN {X 0,Y 269.384,Z 1011.222,A -85,B 0,C 180,E1 11838.363,E2 11838.363} C_VEL
LIN {X 0,Y 258.376,Z 1023.94,A -85,B 0,C 180,E1 11834.153,E2 11834.153} C_VEL
LIN {X 0,Y 248.504,Z 1034.966,A -85,B 0,C 180,E1 11829.474,E2 11829.474} C_VEL
LIN {X 0,Y 239.962,Z 1044.827,A -85,B 0,C 180,E1 11824.231,E2 11824.231} C_VEL
LIN {X 0,Y 233.287,Z 1052.746,A -85,B 0,C 180,E1 11818.688,E2 11818.688} C_VEL
LIN {X 0,Y 228.711,Z 1058.908,A -85,B 0,C 180,E1 11813.17,E2 11813.17} C_VEL
LIN {X 0,Y 225.515,Z 1064.125,A -85,B 0,C 180,E1 11806.723,E2 11806.723} C_VEL
LIN {X 0,Y 224.312,Z 1066.99,A -85,B 0,C 180,E1 11801.572,E2 11801.572} C_VEL
LIN {X 0,Y 223.979,Z 1068.777,A -85,B 0,C 180,E1 11796.408,E2 11796.408} C_VEL
LIN {X 0,Y 224.01,Z 1069.469,A -85,B 0,C 180,E1 11791.279,E2 11791.279} C_VEL
LIN {X 0,Y 223.991,Z 1069.015,A -85,B 0,C 180,E1 11786.417,E2 11786.417} C_VEL
LIN {X 0,Y 224.053,Z 1067.383,A -85,B 0,C 180,E1 11781.273,E2 11781.273} C_VEL
LIN {X 0,Y 224.71,Z 1064.64,A -85,B 0,C 180,E1 11776.097,E2 11776.097} C_VEL
LIN {X 0,Y 226.6,Z 1060.347,A -85,B 0,C 180,E1 11770.406,E2 11770.406} C_VEL
LIN {X 0,Y 230.424,Z 1053.913,A -85,B 0,C 180,E1 11764.282,E2 11764.282} C_VEL
LIN {X 0,Y 235.435,Z 1046.841,A -85,B 0,C 180,E1 11759.077,E2 11759.077} C_VEL
LIN {X 0,Y 243.47,Z 1036.499,A -85,B 0,C 180,E1 11753.159,E2 11753.159} C_VEL
LIN {X 0,Y 251.465,Z 1026.59,A -85,B 0,C 180,E1 11748.696,E2 11748.696} C_VEL
LIN {X 0,Y 262.304,Z 1013.248,A -85,B 0,C 180,E1 11743.908,E2 11743.908} C_VEL
LIN {X 0,Y 272.513,Z 1000.343,A -85,B 0,C 180,E1 11740.224,E2 11740.224} C_VEL
LIN {X 0,Y 284.845,Z 984.13,A -85,B 0,C 180,E1 11736.5,E2 11736.5} C_VEL
LIN {X 0,Y 295.676,Z 968.974,A -85,B 0,C 180,E1 11733.706,E2 11733.706} C_VEL
LIN {X 0,Y 307.858,Z 950.808,A -85,B 0,C 180,E1 11730.969,E2 11730.969} C_VEL
LIN {X 0,Y 318.866,Z 932.772,A -85,B 0,C 180,E1 11728.783,E2 11728.783} C_VEL
LIN {X 0,Y 329.909,Z 913.124,A -85,B 0,C 180,E1 11726.821,E2 11726.821} C_VEL
LIN {X 0,Y 340.246,Z 892.323,A -85,B 0,C 180,E1 11725.16,E2 11725.16} C_VEL
LIN {X 0,Y 349.638,Z 871.278,A -85,B 0,C 180,E1 11723.776,E2 11723.776} C_VEL
LIN {X 0,Y 358.028,Z 849.339,A -85,B 0,C 180,E1 11722.63,E2 11722.63} C_VEL
LIN {X 0,Y 364.543,Z 829.829,A -85,B 0,C 180,E1 11721.805,E2 11721.805} C_VEL
LIN {X 0,Y 371.552,Z 804.574,A -85,B 0,C 180,E1 11720.962,E2 11720.962} C_VEL
LIN {X 0,Y 376.275,Z 783.017,A -85,B 0,C 180,E1 11720.412,E2 11720.412} C_VEL
LIN {X 0,Y 380.395,Z 757.375,A -85,B 0,C 180,E1 11719.894,E2 11719.894} C_VEL
LIN {X 0,Y 387.886,Z 678.764,A -85,B 0,C 180,E1 11718.639,E2 11718.639} C_VEL
LIN {X 0,Y 397.206,Z 578.193,A -85,B 0,C 180,E1 11717.054,E2 11717.054} C_VEL
LIN {X 0,Y 393.989,Z 570.875,A -85,B 0,C 180,E1 11715.116,E2 11715.116} C_VEL
LIN {X 0,Y 389.653,Z 562.753,A -85,B 0,C 180,E1 11712.147,E2 11712.147} C_VEL
LIN {X 0,Y 387.019,Z 558.202,A -85,B 0,C 180,E1 11709.968,E2 11709.968} C_VEL
LIN {X 0,Y 384.996,Z 554.581,A -85,B 0,C 180,E1 11707.912,E2 11707.912} C_VEL
LIN {X 0,Y 382.923,Z 550.71,A -85,B 0,C 180,E1 11705.093,E2 11705.093} C_VEL
LIN {X 0,Y 381.159,Z 546.277,A -85,B 0,C 180,E1 11698.647,E2 11698.647} C_VEL
LIN {X 0,Y 383.252,Z 551.234,A -85,B 0,C 180,E1 11691.976,E2 11691.976} C_VEL
LIN {X 0,Y 385.89,Z 556.083,A -85,B 0,C 180,E1 11688.718,E2 11688.718} C_VEL
LIN {X 0,Y 388.626,Z 561.047,A -85,B 0,C 180,E1 11686.232,E2 11686.232} C_VEL
LIN {X 0,Y 392.071,Z 567.186,A -85,B 0,C 180,E1 11683.708,E2 11683.708} C_VEL
LIN {X 0,Y 397.023,Z 576.643,A -85,B 0,C 180,E1 11680.698,E2 11680.698} C_VEL
LIN {X 0,Y 397.235,Z 577.499,A -85,B 0,C 180,E1 11680.556,E2 11680.556} C_VEL
LIN {X 0,Y 381.103,Z 748.566,A -85,B 0,C 180,E1 11677.881,E2 11677.881} C_VEL
LIN {X 0,Y 377.011,Z 774.925,A -85,B 0,C 180,E1 11677.336,E2 11677.336} C_VEL
LIN {X 0,Y 372.563,Z 795.837,A -85,B 0,C 180,E1 11676.766,E2 11676.766} C_VEL
LIN {X 0,Y 365.89,Z 820.783,A -85,B 0,C 180,E1 11675.887,E2 11675.887} C_VEL
LIN {X 0,Y 359.201,Z 841.277,A -85,B 0,C 180,E1 11674.968,E2 11674.968} C_VEL
LIN {X 0,Y 350.7,Z 863.813,A -85,B 0,C 180,E1 11673.725,E2 11673.725} C_VEL
LIN {X 0,Y 341.559,Z 884.422,A -85,B 0,C 180,E1 11672.319,E2 11672.319} C_VEL
LIN {X 0,Y 331.921,Z 903.982,A -85,B 0,C 180,E1 11670.703,E2 11670.703} C_VEL
LIN {X 0,Y 320.748,Z 924.011,A -85,B 0,C 180,E1 11668.667,E2 11668.667} C_VEL
LIN {X 0,Y 310.371,Z 941.03,A -85,B 0,C 180,E1 11666.571,E2 11666.571} C_VEL
LIN {X 0,Y 298.317,Z 959.043,A -85,B 0,C 180,E1 11663.849,E2 11663.849} C_VEL
LIN {X 0,Y 287.709,Z 973.781,A -85,B 0,C 180,E1 11661.121,E2 11661.121} C_VEL
LIN {X 0,Y 275.441,Z 989.761,A -85,B 0,C 180,E1 11657.47,E2 11657.47} C_VEL
LIN {X 0,Y 265.709,Z 1001.804,A -85,B 0,C 180,E1 11654.048,E2 11654.048} C_VEL
LIN {X 0,Y 255.317,Z 1014.345,A -85,B 0,C 180,E1 11649.669,E2 11649.669} C_VEL
LIN {X 0,Y 246.25,Z 1024.988,A -85,B 0,C 180,E1 11644.926,E2 11644.926} C_VEL
LIN {X 0,Y 238.464,Z 1034.429,A -85,B 0,C 180,E1 11639.655,E2 11639.655} C_VEL
LIN {X 0,Y 232.457,Z 1041.978,A -85,B 0,C 180,E1 11634.119,E2 11634.119} C_VEL
LIN {X 0,Y 228.221,Z 1048.067,A -85,B 0,C 180,E1 11628.388,E2 11628.388} C_VEL
LIN {X 0,Y 225.534,Z 1052.657,A -85,B 0,C 180,E1 11622.287,E2 11622.287} C_VEL
LIN {X 0,Y 224.445,Z 1055.317,A -85,B 0,C 180,E1 11617.166,E2 11617.166} C_VEL
LIN {X 0,Y 224.076,Z 1056.938,A -85,B 0,C 180,E1 11612.046,E2 11612.046} C_VEL
LIN {X 0,Y 224.022,Z 1057.518,A -85,B 0,C 180,E1 11606.674,E2 11606.674} C_VEL
LIN {X 0,Y 224.227,Z 1056.838,A -85,B 0,C 180,E1 11601.279,E2 11601.279} C_VEL
LIN {X 0,Y 224.953,Z 1055.147,A -85,B 0,C 180,E1 11596.112,E2 11596.112} C_VEL
LIN {X 0,Y 226.857,Z 1052.087,A -85,B 0,C 180,E1 11590.429,E2 11590.429} C_VEL
LIN {X 0,Y 230.594,Z 1047.079,A -85,B 0,C 180,E1 11584.303,E2 11584.303} C_VEL
LIN {X 0,Y 235.517,Z 1041.292,A -85,B 0,C 180,E1 11579.048,E2 11579.048} C_VEL
LIN {X 0,Y 243.335,Z 1032.69,A -85,B 0,C 180,E1 11573.135,E2 11573.135} C_VEL
LIN {X 0,Y 251.188,Z 1024.22,A -85,B 0,C 180,E1 11568.64,E2 11568.64} C_VEL
LIN {X 0,Y 261.331,Z 1013.301,A -85,B 0,C 180,E1 11564.002,E2 11564.002} C_VEL
LIN {X 0,Y 271.895,Z 1001.438,A -85,B 0,C 180,E1 11560.058,E2 11560.058} C_VEL
LIN {X 0,Y 283.435,Z 988.076,A -85,B 0,C 180,E1 11556.455,E2 11556.455} C_VEL
LIN {X 0,Y 295.45,Z 973.104,A -85,B 0,C 180,E1 11553.248,E2 11553.248} C_VEL
LIN {X 0,Y 306.754,Z 958.132,A -85,B 0,C 180,E1 11550.624,E2 11550.624} C_VEL
LIN {X 0,Y 319.664,Z 939.475,A -85,B 0,C 180,E1 11547.982,E2 11547.982} C_VEL
LIN {X 0,Y 329.702,Z 923.628,A -85,B 0,C 180,E1 11546.145,E2 11546.145} C_VEL
LIN {X 0,Y 341.262,Z 903.562,A -85,B 0,C 180,E1 11544.217,E2 11544.217} C_VEL
LIN {X 0,Y 350.777,Z 884.924,A -85,B 0,C 180,E1 11542.759,E2 11542.759} C_VEL
LIN {X 0,Y 360.324,Z 864.084,A -85,B 0,C 180,E1 11541.408,E2 11541.408} C_VEL
LIN {X 0,Y 369.07,Z 841.614,A -85,B 0,C 180,E1 11540.23,E2 11540.23} C_VEL
LIN {X 0,Y 376.17,Z 820.468,A -85,B 0,C 180,E1 11539.332,E2 11539.332} C_VEL
LIN {X 0,Y 382.899,Z 795.872,A -85,B 0,C 180,E1 11538.513,E2 11538.513} C_VEL
LIN {X 0,Y 387.518,Z 774.707,A -85,B 0,C 180,E1 11537.969,E2 11537.969} C_VEL
LIN {X 0,Y 391.73,Z 747.973,A -85,B 0,C 180,E1 11537.447,E2 11537.447} C_VEL
LIN {X 0,Y 407.604,Z 585.037,A -85,B 0,C 180,E1 11534.965,E2 11534.965} C_VEL
LIN {X 0,Y 403.504,Z 577.084,A -85,B 0,C 180,E1 11532.159,E2 11532.159} C_VEL
LIN {X 0,Y 400.575,Z 571.719,A -85,B 0,C 180,E1 11529.7,E2 11529.7} C_VEL
LIN {X 0,Y 398.739,Z 568.31,A -85,B 0,C 180,E1 11527.783,E2 11527.783} C_VEL
LIN {X 0,Y 396.971,Z 564.739,A -85,B 0,C 180,E1 11525.334,E2 11525.334} C_VEL
LIN {X 0,Y 396.187,Z 564.939,A -85,B 0,C 180,E1 11524.219,E2 11524.219} C_VEL
LIN {X 0,Y 394.357,Z 569.171,A -85,B 0,C 180,E1 11521.132,E2 11521.132} C_VEL
LIN {X 0,Y 394.191,Z 569.196,A -85,B 0,C 180,E1 11520.245,E2 11520.245} C_VEL
LIN {X 0,Y 394.201,Z 568.561,A -85,B 0,C 180,E1 11518.983,E2 11518.983} C_VEL
LIN {X 0,Y 395.985,Z 572.93,A -85,B 0,C 180,E1 11512.966,E2 11512.966} C_VEL
LIN {X 0,Y 398.325,Z 577.571,A -85,B 0,C 180,E1 11509.88,E2 11509.88} C_VEL
LIN {X 0,Y 400.85,Z 582.375,A -85,B 0,C 180,E1 11507.466,E2 11507.466} C_VEL
LIN {X 0,Y 403.733,Z 588.041,A -85,B 0,C 180,E1 11505.221,E2 11505.221} C_VEL
LIN {X 0,Y 404.955,Z 591.395,A -85,B 0,C 180,E1 11504.314,E2 11504.314} C_VEL
LIN {X 0,Y 388.666,Z 755.37,A -85,B 0,C 180,E1 11501.838,E2 11501.838} C_VEL
LIN {X 0,Y 384.319,Z 781.902,A -85,B 0,C 180,E1 11501.343,E2 11501.343} C_VEL
LIN {X 0,Y 379.456,Z 803.341,A -85,B 0,C 180,E1 11500.844,E2 11500.844} C_VEL
LIN {X 0,Y 372.227,Z 828.54,A -85,B 0,C 180,E1 11500.082,E2 11500.082} C_VEL
LIN {X 0,Y 365.063,Z 849.096,A -85,B 0,C 180,E1 11499.285,E2 11499.285} C_VEL
LIN {X 0,Y 355.947,Z 871.697,A -85,B 0,C 180,E1 11498.188,E2 11498.188} C_VEL
LIN {X 0,Y 346.182,Z 892.468,A -85,B 0,C 180,E1 11496.917,E2 11496.917} C_VEL
LIN {X 0,Y 335.432,Z 912.933,A -85,B 0,C 180,E1 11495.392,E2 11495.392} C_VEL
LIN {X 0,Y 323.799,Z 932.413,A -85,B 0,C 180,E1 11493.575,E2 11493.575} C_VEL
LIN {X 0,Y 312.182,Z 950.261,A -85,B 0,C 180,E1 11491.546,E2 11491.546} C_VEL
LIN {X 0,Y 299.551,Z 967.837,A -85,B 0,C 180,E1 11489.066,E2 11489.066} C_VEL
LIN {X 0,Y 288.164,Z 982.576,A -85,B 0,C 180,E1 11486.516,E2 11486.516} C_VEL
LIN {X 0,Y 274.431,Z 999.159,A -85,B 0,C 180,E1 11482.933,E2 11482.933} C_VEL
LIN {X 0,Y 263.197,Z 1011.954,A -85,B 0,C 180,E1 11479.447,E2 11479.447} C_VEL
LIN {X 0,Y 250.983,Z 1025.361,A -85,B 0,C 180,E1 11474.835,E2 11474.835} C_VEL
LIN {X 0,Y 241.502,Z 1035.524,A -85,B 0,C 180,E1 11470.375,E2 11470.375} C_VEL
LIN {X 0,Y 232.464,Z 1045.385,A -85,B 0,C 180,E1 11464.895,E2 11464.895} C_VEL
LIN {X 0,Y 225.807,Z 1052.876,A -85,B 0,C 180,E1 11459.44,E2 11459.44} C_VEL
LIN {X 0,Y 220.639,Z 1059.497,A -85,B 0,C 180,E1 11453.22,E2 11453.22} C_VEL
LIN {X 0,Y 217.522,Z 1064.242,A -85,B 0,C 180,E1 11446.834,E2 11446.834} C_VEL
LIN {X 0,Y 216.293,Z 1067.025,A -85,B 0,C 180,E1 11441.464,E2 11441.464} C_VEL
LIN {X 0,Y 215.98,Z 1068.863,A -85,B 0,C 180,E1 11435.522,E2 11435.522} C_VEL
LIN {X 0,Y 216.025,Z 1069.208,A -85,B 0,C 180,E1 11430.265,E2 11430.265} C_VEL
LIN {X 0,Y 215.988,Z 1068.582,A -85,B 0,C 180,E1 11425.486,E2 11425.486} C_VEL
LIN {X 0,Y 216.102,Z 1066.917,A -85,B 0,C 180,E1 11420.412,E2 11420.412} C_VEL
LIN {X 0,Y 216.871,Z 1064.236,A -85,B 0,C 180,E1 11415.311,E2 11415.311} C_VEL
LIN {X 0,Y 219.153,Z 1059.671,A -85,B 0,C 180,E1 11409.153,E2 11409.153} C_VEL
LIN {X 0,Y 223.315,Z 1053.221,A -85,B 0,C 180,E1 11403.002,E2 11403.002} C_VEL
LIN {X 0,Y 229.108,Z 1045.667,A -85,B 0,C 180,E1 11397.385,E2 11397.385} C_VEL
LIN {X 0,Y 237.26,Z 1035.745,A -85,B 0,C 180,E1 11391.72,E2 11391.72} C_VEL
LIN {X 0,Y 245.743,Z 1025.772,A -85,B 0,C 180,E1 11387.196,E2 11387.196} C_VEL
LIN {X 0,Y 257.141,Z 1012.292,A -85,B 0,C 180,E1 11382.37,E2 11382.37} C_VEL
LIN {X 0,Y 267.758,Z 999.38,A -85,B 0,C 180,E1 11378.697,E2 11378.697} C_VEL
LIN {X 0,Y 280.637,Z 982.934,A -85,B 0,C 180,E1 11374.968,E2 11374.968} C_VEL
LIN {X 0,Y 291.856,Z 967.687,A -85,B 0,C 180,E1 11372.198,E2 11372.198} C_VEL
LIN {X 0,Y 305.139,Z 948.186,A -85,B 0,C 180,E1 11369.351,E2 11369.351} C_VEL
LIN {X 0,Y 315.369,Z 931.769,A -85,B 0,C 180,E1 11367.408,E2 11367.408} C_VEL
LIN {X 0,Y 327.106,Z 911.145,A -85,B 0,C 180,E1 11365.408,E2 11365.408} C_VEL
LIN {X 0,Y 336.859,Z 891.881,A -85,B 0,C 180,E1 11363.904,E2 11363.904} C_VEL
LIN {X 0,Y 346.84,Z 869.832,A -85,B 0,C 180,E1 11362.489,E2 11362.489} C_VEL
LIN {X 0,Y 355.392,Z 847.669,A -85,B 0,C 180,E1 11361.367,E2 11361.367} C_VEL
LIN {X 0,Y 363.073,Z 824.71,A -85,B 0,C 180,E1 11360.441,E2 11360.441} C_VEL
LIN {X 0,Y 369.397,Z 801.15,A -85,B 0,C 180,E1 11359.715,E2 11359.715} C_VEL
LIN {X 0,Y 374.38,Z 778.046,A -85,B 0,C 180,E1 11359.159,E2 11359.159} C_VEL
LIN {X 0,Y 378.077,Z 753.063,A -85,B 0,C 180,E1 11358.686,E2 11358.686} C_VEL
LIN {X 0,Y 394.351,Z 583.045,A -85,B 0,C 180,E1 11356.044,E2 11356.044} C_VEL
LIN {X 0,Y 391.902,Z 577.444,A -85,B 0,C 180,E1 11354.48,E2 11354.48} C_VEL
LIN {X 0,Y 387.716,Z 569.519,A -85,B 0,C 180,E1 11351.454,E2 11351.454} C_VEL
LIN {X 0,Y 385.551,Z 565.623,A -85,B 0,C 180,E1 11349.554,E2 11349.554} C_VEL
LIN {X 0,Y 383.879,Z 562.467,A -85,B 0,C 180,E1 11347.784,E2 11347.784} C_VEL
LIN {X 0,Y 381.85,Z 558.59,A -85,B 0,C 180,E1 11344.957,E2 11344.957} C_VEL
LIN {X 0,Y 380.177,Z 554.278,A -85,B 0,C 180,E1 11338.644,E2 11338.644} C_VEL
LIN {X 0,Y 382.169,Z 559.167,A -85,B 0,C 180,E1 11332.105,E2 11332.105} C_VEL
LIN {X 0,Y 384.686,Z 563.928,A -85,B 0,C 180,E1 11328.91,E2 11328.91} C_VEL
LIN {X 0,Y 387.275,Z 568.76,A -85,B 0,C 180,E1 11326.487,E2 11326.487} C_VEL
LIN {X 0,Y 390.585,Z 574.877,A -85,B 0,C 180,E1 11323.988,E2 11323.988} C_VEL
LIN {X 0,Y 394.342,Z 582.297,A -85,B 0,C 180,E1 11321.588,E2 11321.588} C_VEL
LIN {X 0,Y 378.296,Z 748.83,A -85,B 0,C 180,E1 11319.011,E2 11319.011} C_VEL
LIN {X 0,Y 374.118,Z 775.234,A -85,B 0,C 180,E1 11318.474,E2 11318.474} C_VEL
LIN {X 0,Y 369.59,Z 796.141,A -85,B 0,C 180,E1 11317.914,E2 11317.914} C_VEL
LIN {X 0,Y 363.105,Z 820.102,A -85,B 0,C 180,E1 11317.09,E2 11317.09} C_VEL
LIN {X 0,Y 356.291,Z 840.703,A -85,B 0,C 180,E1 11316.189,E2 11316.189} C_VEL
LIN {X 0,Y 347.935,Z 862.643,A -85,B 0,C 180,E1 11315.011,E2 11315.011} C_VEL
LIN {X 0,Y 338.291,Z 884.075,A -85,B 0,C 180,E1 11313.583,E2 11313.583} C_VEL
LIN {X 0,Y 328.842,Z 902.891,A -85,B 0,C 180,E1 11312.062,E2 11312.062} C_VEL
LIN {X 0,Y 317.357,Z 923.205,A -85,B 0,C 180,E1 11310.047,E2 11310.047} C_VEL
LIN {X 0,Y 307.054,Z 939.742,A -85,B 0,C 180,E1 11308.054,E2 11308.054} C_VEL
LIN {X 0,Y 294.341,Z 958.4,A -85,B 0,C 180,E1 11305.294,E2 11305.294} C_VEL
LIN {X 0,Y 283.827,Z 972.616,A -85,B 0,C 180,E1 11302.703,E2 11302.703} C_VEL
LIN {X 0,Y 271.761,Z 988.016,A -85,B 0,C 180,E1 11299.282,E2 11299.282} C_VEL
LIN {X 0,Y 260.571,Z 1001.343,A -85,B 0,C 180,E1 11295.54,E2 11295.54} C_VEL
LIN {X 0,Y 249.83,Z 1013.835,A -85,B 0,C 180,E1 11291.198,E2 11291.198} C_VEL
LIN {X 0,Y 240.003,Z 1024.826,A -85,B 0,C 180,E1 11286.27,E2 11286.27} C_VEL
LIN {X 0,Y 231.738,Z 1034.345,A -85,B 0,C 180,E1 11280.894,E2 11280.894} C_VEL
LIN {X 0,Y 225.118,Z 1042.167,A -85,B 0,C 180,E1 11275.028,E2 11275.028} C_VEL
LIN {X 0,Y 220.545,Z 1048.322,A -85,B 0,C 180,E1 11269.052,E2 11269.052} C_VEL
LIN {X 0,Y 217.661,Z 1052.896,A -85,B 0,C 180,E1 11262.738,E2 11262.738} C_VEL
LIN {X 0,Y 216.482,Z 1055.548,A -85,B 0,C 180,E1 11257.431,E2 11257.431} C_VEL
LIN {X 0,Y 216.081,Z 1057.161,A -85,B 0,C 180,E1 11252.121,E2 11252.121} C_VEL
LIN {X 0,Y 216.023,Z 1057.746,A -85,B 0,C 180,E1 11246.816,E2 11246.816} C_VEL
LIN {X 0,Y 216.234,Z 1057.109,A -85,B 0,C 180,E1 11241.223,E2 11241.223} C_VEL
LIN {X 0,Y 217.003,Z 1055.456,A -85,B 0,C 180,E1 11235.865,E2 11235.865} C_VEL
LIN {X 0,Y 218.92,Z 1052.565,A -85,B 0,C 180,E1 11230.201,E2 11230.201} C_VEL
LIN {X 0,Y 222.985,Z 1047.508,A -85,B 0,C 180,E1 11223.645,E2 11223.645} C_VEL
LIN {X 0,Y 228.181,Z 1041.755,A -85,B 0,C 180,E1 11218.224,E2 11218.224} C_VEL
LIN {X 0,Y 236.021,Z 1033.63,A -85,B 0,C 180,E1 11212.393,E2 11212.393} C_VEL
LIN {X 0,Y 244.575,Z 1024.825,A -85,B 0,C 180,E1 11207.58,E2 11207.58} C_VEL
LIN {X 0,Y 255.125,Z 1013.998,A -85,B 0,C 180,E1 11202.87,E2 11202.87} C_VEL
LIN {X 0,Y 266.567,Z 1001.642,A -85,B 0,C 180,E1 11198.721,E2 11198.721} C_VEL
LIN {X 0,Y 278.914,Z 987.844,A -85,B 0,C 180,E1 11195.001,E2 11195.001} C_VEL
LIN {X 0,Y 291.601,Z 972.449,A -85,B 0,C 180,E1 11191.747,E2 11191.747} C_VEL
LIN {X 0,Y 304.417,Z 955.9,A -85,B 0,C 180,E1 11188.914,E2 11188.914} C_VEL
LIN {X 0,Y 316.764,Z 938.223,A -85,B 0,C 180,E1 11186.506,E2 11186.506} C_VEL
LIN {X 0,Y 328.092,Z 920.623,A -85,B 0,C 180,E1 11184.535,E2 11184.535} C_VEL
LIN {X 0,Y 339.836,Z 900.107,A -85,B 0,C 180,E1 11182.671,E2 11182.671} C_VEL
LIN {X 0,Y 349.323,Z 881.65,A -85,B 0,C 180,E1 11181.299,E2 11181.299} C_VEL
LIN {X 0,Y 359.482,Z 859.074,A -85,B 0,C 180,E1 11179.925,E2 11179.925} C_VEL
LIN {X 0,Y 366.898,Z 840.001,A -85,B 0,C 180,E1 11178.975,E2 11178.975} C_VEL
LIN {X 0,Y 374.661,Z 816.827,A -85,B 0,C 180,E1 11178.034,E2 11178.034} C_VEL
LIN {X 0,Y 380.859,Z 793.719,A -85,B 0,C 180,E1 11177.307,E2 11177.307} C_VEL
LIN {X 0,Y 386.033,Z 769.656,A -85,B 0,C 180,E1 11176.723,E2 11176.723} C_VEL
LIN {X 0,Y 389.616,Z 745.218,A -85,B 0,C 180,E1 11176.282,E2 11176.282} C_VEL
LIN {X 0,Y 404.922,Z 590.346,A -85,B 0,C 180,E1 11173.932,E2 11173.932} C_VEL
LIN {X 0,Y 401.251,Z 583.168,A -85,B 0,C 180,E1 11171.208,E2 11171.208} C_VEL
LIN {X 0,Y 398.992,Z 578.889,A -85,B 0,C 180,E1 11169.157,E2 11169.157} C_VEL
LIN {X 0,Y 397.505,Z 576.015,A -85,B 0,C 180,E1 11167.516,E2 11167.516} C_VEL
LIN {X 0,Y 395.726,Z 572.441,A -85,B 0,C 180,E1 11164.928,E2 11164.928} C_VEL
LIN {X 0,Y 394.191,Z 569.196,A -85,B 0,C 180,E1 11160.245,E2 11160.245} C_VEL
LIN {X 0,Y 394.072,Z 569.689,A -85,B 0,C 180,E1 11159.608,E2 11159.608} C_VEL
LIN {X 0,Y 393.674,Z 572.986,A -85,B 0,C 180,E1 11158.623,E2 11158.623} C_VEL
LIN {X 0,Y 393.316,Z 577.058,A -85,B 0,C 180,E1 11157.536,E2 11157.536} C_VEL
LIN {X 0,Y 393.327,Z 577.972,A -85,B 0,C 180,E1 11156.997,E2 11156.997} C_VEL
LIN {X 0,Y 394.911,Z 580.859,A -85,B 0,C 180,E1 11153.092,E2 11153.092} C_VEL
LIN {X 0,Y 397.137,Z 585.407,A -85,B 0,C 180,E1 11150.069,E2 11150.069} C_VEL
LIN {X 0,Y 399.686,Z 590.391,A -85,B 0,C 180,E1 11147.576,E2 11147.576} C_VEL
LIN {X 0,Y 402.368,Z 595.995,A -85,B 0,C 180,E1 11145.427,E2 11145.427} C_VEL
LIN {X 0,Y 402.437,Z 596.658,A -85,B 0,C 180,E1 11145.339,E2 11145.339} C_VEL
LIN {X 0,Y 386.359,Z 755.249,A -85,B 0,C 180,E1 11142.975,E2 11142.975} C_VEL
LIN {X 0,Y 381.94,Z 781.772,A -85,B 0,C 180,E1 11142.489,E2 11142.489} C_VEL
LIN {X 0,Y 377,Z 803.226,A -85,B 0,C 180,E1 11142.003,E2 11142.003} C_VEL
LIN {X 0,Y 369.57,Z 828.679,A -85,B 0,C 180,E1 11141.252,E2 11141.252} C_VEL
LIN {X 0,Y 362.338,Z 849.079,A -85,B 0,C 180,E1 11140.48,E2 11140.48} C_VEL
LIN {X 0,Y 352.609,Z 872.629,A -85,B 0,C 180,E1 11139.354,E2 11139.354} C_VEL
LIN {X 0,Y 343.092,Z 892.475,A -85,B 0,C 180,E1 11138.159,E2 11138.159} C_VEL
LIN {X 0,Y 332.136,Z 912.908,A -85,B 0,C 180,E1 11136.664,E2 11136.664} C_VEL
LIN {X 0,Y 320.172,Z 932.497,A -85,B 0,C 180,E1 11134.867,E2 11134.867} C_VEL
LIN {X 0,Y 307.996,Z 950.753,A -85,B 0,C 180,E1 11132.813,E2 11132.813} C_VEL
LIN {X 0,Y 294.932,Z 968.373,A -85,B 0,C 180,E1 11130.332,E2 11130.332} C_VEL
LIN {X 0,Y 283.199,Z 983.106,A -85,B 0,C 180,E1 11127.782,E2 11127.782} C_VEL
LIN {X 0,Y 269.54,Z 999.036,A -85,B 0,C 180,E1 11124.332,E2 11124.332} C_VEL
LIN {X 0,Y 258.487,Z 1011.181,A -85,B 0,C 180,E1 11121.034,E2 11121.034} C_VEL
LIN {X 0,Y 246.232,Z 1024.161,A -85,B 0,C 180,E1 11116.625,E2 11116.625} C_VEL
LIN {X 0,Y 235.946,Z 1034.651,A -85,B 0,C 180,E1 11112.034,E2 11112.034} C_VEL
LIN {X 0,Y 226.454,Z 1044.49,A -85,B 0,C 180,E1 11106.59,E2 11106.59} C_VEL
LIN {X 0,Y 218.925,Z 1052.388,A -85,B 0,C 180,E1 11100.766,E2 11100.766} C_VEL
LIN {X 0,Y 213.517,Z 1058.736,A -85,B 0,C 180,E1 11094.702,E2 11094.702} C_VEL
LIN {X 0,Y 209.917,Z 1063.715,A -85,B 0,C 180,E1 11088.036,E2 11088.036} C_VEL
LIN {X 0,Y 208.437,Z 1066.587,A -85,B 0,C 180,E1 11082.467,E2 11082.467} C_VEL
LIN {X 0,Y 207.988,Z 1068.365,A -85,B 0,C 180,E1 11076.903,E2 11076.903} C_VEL
LIN {X 0,Y 208.013,Z 1069.047,A -85,B 0,C 180,E1 11071.377,E2 11071.377} C_VEL
LIN {X 0,Y 207.992,Z 1068.569,A -85,B 0,C 180,E1 11066.141,E2 11066.141} C_VEL
LIN {X 0,Y 208.09,Z 1066.922,A -85,B 0,C 180,E1 11060.597,E2 11060.597} C_VEL
LIN {X 0,Y 208.923,Z 1064.162,A -85,B 0,C 180,E1 11055.023,E2 11055.023} C_VEL
LIN {X 0,Y 211.253,Z 1059.78,A -85,B 0,C 180,E1 11048.818,E2 11048.818} C_VEL
LIN {X 0,Y 215.751,Z 1053.27,A -85,B 0,C 180,E1 11042.274,E2 11042.274} C_VEL
LIN {X 0,Y 221.374,Z 1046.302,A -85,B 0,C 180,E1 11036.871,E2 11036.871} C_VEL
LIN {X 0,Y 230.388,Z 1035.929,A -85,B 0,C 180,E1 11030.681,E2 11030.681} C_VEL
LIN {X 0,Y 239.234,Z 1026.005,A -85,B 0,C 180,E1 11026.068,E2 11026.068} C_VEL
LIN {X 0,Y 251.067,Z 1012.628,A -85,B 0,C 180,E1 11021.175,E2 11021.175} C_VEL
LIN {X 0,Y 261.443,Z 1000.486,A -85,B 0,C 180,E1 11017.658,E2 11017.658} C_VEL
LIN {X 0,Y 274.013,Z 985.169,A -85,B 0,C 180,E1 11014.072,E2 11014.072} C_VEL
LIN {X 0,Y 286.148,Z 969.215,A -85,B 0,C 180,E1 11011.118,E2 11011.118} C_VEL
LIN {X 0,Y 298.699,Z 951.636,A -85,B 0,C 180,E1 11008.474,E2 11008.474} C_VEL
LIN {X 0,Y 310.577,Z 933.16,A -85,B 0,C 180,E1 11006.26,E2 11006.26} C_VEL
LIN {X 0,Y 322.111,Z 913.631,A -85,B 0,C 180,E1 11004.345,E2 11004.345} C_VEL
LIN {X 0,Y 332.832,Z 893.076,A -85,B 0,C 180,E1 11002.738,E2 11002.738} C_VEL
LIN {X 0,Y 342.167,Z 873.069,A -85,B 0,C 180,E1 11001.451,E2 11001.451} C_VEL
LIN {X 0,Y 351.268,Z 850.561,A -85,B 0,C 180,E1 11000.294,E2 11000.294} C_VEL
LIN {X 0,Y 358.056,Z 831.097,A -85,B 0,C 180,E1 10999.494,E2 10999.494} C_VEL
LIN {X 0,Y 365.017,Z 807.553,A -85,B 0,C 180,E1 10998.718,E2 10998.718} C_VEL
LIN {X 0,Y 370.365,Z 784.322,A -85,B 0,C 180,E1 10998.138,E2 10998.138} C_VEL
LIN {X 0,Y 374.65,Z 759.685,A -85,B 0,C 180,E1 10997.646,E2 10997.646} C_VEL
LIN {X 0,Y 379.883,Z 708.542,A -85,B 0,C 180,E1 10996.836,E2 10996.836} C_VEL
LIN {X 0,Y 391.56,Z 587.862,A -85,B 0,C 180,E1 10994.987,E2 10994.987} C_VEL
LIN {X 0,Y 388.687,Z 581.723,A -85,B 0,C 180,E1 10993.008,E2 10993.008} C_VEL
LIN {X 0,Y 384.958,Z 574.441,A -85,B 0,C 180,E1 10989.946,E2 10989.946} C_VEL
LIN {X 0,Y 382.634,Z 570.172,A -85,B 0,C 180,E1 10987.508,E2 10987.508} C_VEL
LIN {X 0,Y 380.687,Z 566.377,A -85,B 0,C 180,E1 10984.67,E2 10984.67} C_VEL
LIN {X 0,Y 379.195,Z 562.276,A -85,B 0,C 180,E1 10978.64,E2 10978.64} C_VEL
LIN {X 0,Y 381.047,Z 566.98,A -85,B 0,C 180,E1 10972.309,E2 10972.309} C_VEL
LIN {X 0,Y 383.419,Z 571.626,A -85,B 0,C 180,E1 10969.178,E2 10969.178} C_VEL
LIN {X 0,Y 385.933,Z 576.471,A -85,B 0,C 180,E1 10966.745,E2 10966.745} C_VEL
LIN {X 0,Y 389.259,Z 582.878,A -85,B 0,C 180,E1 10964.162,E2 10964.162} C_VEL
LIN {X 0,Y 391.526,Z 587.637,A -85,B 0,C 180,E1 10962.628,E2 10962.628} C_VEL
LIN {X 0,Y 375.637,Z 749.094,A -85,B 0,C 180,E1 10960.158,E2 10960.158} C_VEL
LIN {X 0,Y 371.401,Z 775.414,A -85,B 0,C 180,E1 10959.632,E2 10959.632} C_VEL
LIN {X 0,Y 366.788,Z 796.366,A -85,B 0,C 180,E1 10959.083,E2 10959.083} C_VEL
LIN {X 0,Y 360.072,Z 820.693,A -85,B 0,C 180,E1 10958.261,E2 10958.261} C_VEL
LIN {X 0,Y 353.14,Z 841.25,A -85,B 0,C 180,E1 10957.375,E2 10957.375} C_VEL
LIN {X 0,Y 344.606,Z 863.202,A -85,B 0,C 180,E1 10956.214,E2 10956.214} C_VEL
LIN {X 0,Y 334.798,Z 884.529,A -85,B 0,C 180,E1 10954.813,E2 10954.813} C_VEL
LIN {X 0,Y 324.731,Z 904.123,A -85,B 0,C 180,E1 10953.246,E2 10953.246} C_VEL
LIN {X 0,Y 313.167,Z 923.993,A -85,B 0,C 180,E1 10951.282,E2 10951.282} C_VEL
LIN {X 0,Y 302.44,Z 940.759,A -85,B 0,C 180,E1 10949.269,E2 10949.269} C_VEL
LIN {X 0,Y 289.803,Z 958.756,A -85,B 0,C 180,E1 10946.611,E2 10946.611} C_VEL
LIN {X 0,Y 278.691,Z 973.331,A -85,B 0,C 180,E1 10943.956,E2 10943.956} C_VEL
LIN {X 0,Y 266.527,Z 988.339,A -85,B 0,C 180,E1 10940.608,E2 10940.608} C_VEL
LIN {X 0,Y 254.93,Z 1001.657,A -85,B 0,C 180,E1 10936.847,E2 10936.847} C_VEL
LIN {X 0,Y 243.96,Z 1013.904,A -85,B 0,C 180,E1 10932.552,E2 10932.552} C_VEL
LIN {X 0,Y 233.898,Z 1024.664,A -85,B 0,C 180,E1 10927.684,E2 10927.684} C_VEL
LIN {X 0,Y 225.465,Z 1033.834,A -85,B 0,C 180,E1 10922.453,E2 10922.453} C_VEL
LIN {X 0,Y 218.219,Z 1041.913,A -85,B 0,C 180,E1 10916.389,E2 10916.389} C_VEL
LIN {X 0,Y 213.595,Z 1047.586,A -85,B 0,C 180,E1 10910.841,E2 10910.841} C_VEL
LIN {X 0,Y 209.997,Z 1052.826,A -85,B 0,C 180,E1 10903.773,E2 10903.773} C_VEL
LIN {X 0,Y 208.607,Z 1055.559,A -85,B 0,C 180,E1 10898.267,E2 10898.267} C_VEL
LIN {X 0,Y 208.115,Z 1057.186,A -85,B 0,C 180,E1 10893.029,E2 10893.029} C_VEL
LIN {X 0,Y 208.016,Z 1057.88,A -85,B 0,C 180,E1 10887.796,E2 10887.796} C_VEL
LIN {X 0,Y 208.182,Z 1057.575,A -85,B 0,C 180,E1 10881.993,E2 10881.993} C_VEL
LIN {X 0,Y 208.993,Z 1055.875,A -85,B 0,C 180,E1 10875.877,E2 10875.877} C_VEL
LIN {X 0,Y 210.945,Z 1053.094,A -85,B 0,C 180,E1 10870.045,E2 10870.045} C_VEL
LIN {X 0,Y 215.281,Z 1048.082,A -85,B 0,C 180,E1 10863.096,E2 10863.096} C_VEL
LIN {X 0,Y 220.897,Z 1042.216,A -85,B 0,C 180,E1 10857.345,E2 10857.345} C_VEL
LIN {X 0,Y 229.132,Z 1034.175,A -85,B 0,C 180,E1 10851.364,E2 10851.364} C_VEL
LIN {X 0,Y 238.514,Z 1024.975,A -85,B 0,C 180,E1 10846.235,E2 10846.235} C_VEL
LIN {X 0,Y 249.555,Z 1014.133,A -85,B 0,C 180,E1 10841.475,E2 10841.475} C_VEL
LIN {X 0,Y 261.467,Z 1001.766,A -85,B 0,C 180,E1 10837.305,E2 10837.305} C_VEL
LIN {X 0,Y 273.934,Z 988.303,A -85,B 0,C 180,E1 10833.672,E2 10833.672} C_VEL
LIN {X 0,Y 286.656,Z 973.382,A -85,B 0,C 180,E1 10830.507,E2 10830.507} C_VEL
LIN {X 0,Y 298.705,Z 958.289,A -85,B 0,C 180,E1 10827.906,E2 10827.906} C_VEL
LIN {X 0,Y 312.054,Z 939.937,A -85,B 0,C 180,E1 10825.366,E2 10825.366} C_VEL
LIN {X 0,Y 323.215,Z 923.089,A -85,B 0,C 180,E1 10823.473,E2 10823.473} C_VEL
LIN {X 0,Y 335.885,Z 901.738,A -85,B 0,C 180,E1 10821.522,E2 10821.522} C_VEL
LIN {X 0,Y 345.221,Z 884.06,A -85,B 0,C 180,E1 10820.211,E2 10820.211} C_VEL
LIN {X 0,Y 355.441,Z 862.284,A -85,B 0,C 180,E1 10818.875,E2 10818.875} C_VEL
LIN {X 0,Y 363.501,Z 842.146,A -85,B 0,C 180,E1 10817.871,E2 10817.871} C_VEL
LIN {X 0,Y 371.133,Z 820.134,A -85,B 0,C 180,E1 10816.976,E2 10816.976} C_VEL
LIN {X 0,Y 377.943,Z 795.836,A -85,B 0,C 180,E1 10816.207,E2 10816.207} C_VEL
LIN {X 0,Y 382.796,Z 774.16,A -85,B 0,C 180,E1 10815.679,E2 10815.679} C_VEL
LIN {X 0,Y 386.985,Z 748.089,A -85,B 0,C 180,E1 10815.193,E2 10815.193} C_VEL
LIN {X 0,Y 402.406,Z 595.907,A -85,B 0,C 180,E1 10812.922,E2 10812.922} C_VEL
LIN {X 0,Y 399.341,Z 589.769,A -85,B 0,C 180,E1 10810.459,E2 10810.459} C_VEL
LIN {X 0,Y 396.711,Z 584.355,A -85,B 0,C 180,E1 10807.75,E2 10807.75} C_VEL
LIN {X 0,Y 394.576,Z 580.237,A -85,B 0,C 180,E1 10804.651,E2 10804.651} C_VEL
LIN {X 0,Y 393.231,Z 576.445,A -85,B 0,C 180,E1 10799.126,E2 10799.126} C_VEL
LIN {X 0,Y 393.327,Z 577.972,A -85,B 0,C 180,E1 10796.997,E2 10796.997} C_VEL
LIN {X 0,Y 393.472,Z 579.728,A -85,B 0,C 180,E1 10795.893,E2 10795.893} C_VEL
LIN {X 0,Y 394.13,Z 589.269,A -85,B 0,C 180,E1 10792.752,E2 10792.752} C_VEL
LIN {X 0,Y 394.497,Z 590.432,A -85,B 0,C 180,E1 10792.124,E2 10792.124} C_VEL
LIN {X 0,Y 395.894,Z 593.101,A -85,B 0,C 180,E1 10790.331,E2 10790.331} C_VEL
LIN {X 0,Y 398.364,Z 598.093,A -85,B 0,C 180,E1 10787.828,E2 10787.828} C_VEL
LIN {X 0,Y 400.05,Z 601.908,A -85,B 0,C 180,E1 10786.377,E2 10786.377} C_VEL
LIN {X 0,Y 384.214,Z 755.061,A -85,B 0,C 180,E1 10784.127,E2 10784.127} C_VEL
LIN {X 0,Y 379.735,Z 781.548,A -85,B 0,C 180,E1 10783.652,E2 10783.652} C_VEL
LIN {X 0,Y 374.706,Z 803.088,A -85,B 0,C 180,E1 10783.177,E2 10783.177} C_VEL
LIN {X 0,Y 367.504,Z 827.537,A -85,B 0,C 180,E1 10782.483,E2 10782.483} C_VEL
LIN {X 0,Y 359.857,Z 848.846,A -85,B 0,C 180,E1 10781.701,E2 10781.701} C_VEL
LIN {X 0,Y 350.274,Z 871.762,A -85,B 0,C 180,E1 10780.638,E2 10780.638} C_VEL
LIN {X 0,Y 340.585,Z 891.671,A -85,B 0,C 180,E1 10779.475,E2 10779.475} C_VEL
LIN {X 0,Y 329.416,Z 912.179,A -85,B 0,C 180,E1 10778.017,E2 10778.017} C_VEL
LIN {X 0,Y 317.283,Z 931.705,A -85,B 0,C 180,E1 10776.275,E2 10776.275} C_VEL
LIN {X 0,Y 305.781,Z 948.621,A -85,B 0,C 180,E1 10774.429,E2 10774.429} C_VEL
LIN {X 0,Y 292.224,Z 966.7,A -85,B 0,C 180,E1 10771.981,E2 10771.981} C_VEL
LIN {X 0,Y 279.875,Z 981.832,A -85,B 0,C 180,E1 10769.429,E2 10769.429} C_VEL
LIN {X 0,Y 265.479,Z 998.208,A -85,B 0,C 180,E1 10765.955,E2 10765.955} C_VEL
LIN {X 0,Y 253.374,Z 1011.049,A -85,B 0,C 180,E1 10762.486,E2 10762.486} C_VEL
LIN {X 0,Y 240.617,Z 1024.011,A -85,B 0,C 180,E1 10758.059,E2 10758.059} C_VEL
LIN {X 0,Y 229.819,Z 1034.529,A -85,B 0,C 180,E1 10753.399,E2 10753.399} C_VEL
LIN {X 0,Y 219.857,Z 1044.319,A -85,B 0,C 180,E1 10747.877,E2 10747.877} C_VEL
LIN {X 0,Y 211.714,Z 1052.364,A -85,B 0,C 180,E1 10741.776,E2 10741.776} C_VEL
LIN {X 0,Y 205.808,Z 1058.873,A -85,B 0,C 180,E1 10735.311,E2 10735.311} C_VEL
LIN {X 0,Y 202.037,Z 1063.683,A -85,B 0,C 180,E1 10728.466,E2 10728.466} C_VEL
LIN {X 0,Y 200.463,Z 1066.504,A -85,B 0,C 180,E1 10722.678,E2 10722.678} C_VEL
LIN {X 0,Y 199.982,Z 1068.373,A -85,B 0,C 180,E1 10716.315,E2 10716.315} C_VEL
LIN {X 0,Y 200.023,Z 1068.819,A -85,B 0,C 180,E1 10710.859,E2 10710.859} C_VEL
LIN {X 0,Y 199.991,Z 1068.276,A -85,B 0,C 180,E1 10705.699,E2 10705.699} C_VEL
LIN {X 0,Y 200.137,Z 1066.573,A -85,B 0,C 180,E1 10699.929,E2 10699.929} C_VEL
LIN {X 0,Y 201.054,Z 1063.923,A -85,B 0,C 180,E1 10694.422,E2 10694.422} C_VEL
LIN {X 0,Y 203.56,Z 1059.605,A -85,B 0,C 180,E1 10688.08,E2 10688.08} C_VEL
LIN {X 0,Y 208.377,Z 1053.128,A -85,B 0,C 180,E1 10681.325,E2 10681.325} C_VEL
LIN {X 0,Y 214.622,Z 1045.879,A -85,B 0,C 180,E1 10675.55,E2 10675.55} C_VEL
LIN {X 0,Y 224.021,Z 1035.644,A -85,B 0,C 180,E1 10669.334,E2 10669.334} C_VEL
LIN {X 0,Y 233.324,Z 1025.711,A -85,B 0,C 180,E1 10664.653,E2 10664.653} C_VEL
LIN {X 0,Y 245.68,Z 1012.315,A -85,B 0,C 180,E1 10659.715,E2 10659.715} C_VEL
LIN {X 0,Y 256.46,Z 1000.167,A -85,B 0,C 180,E1 10656.191,E2 10656.191} C_VEL
LIN {X 0,Y 269.465,Z 984.83,A -85,B 0,C 180,E1 10652.614,E2 10652.614} C_VEL
LIN {X 0,Y 281.973,Z 968.866,A -85,B 0,C 180,E1 10649.683,E2 10649.683} C_VEL
LIN {X 0,Y 294.793,Z 951.371,A -85,B 0,C 180,E1 10647.082,E2 10647.082} C_VEL
LIN {X 0,Y 306.993,Z 932.839,A -85,B 0,C 180,E1 10644.894,E2 10644.894} C_VEL
LIN {X 0,Y 318.827,Z 913.227,A -85,B 0,C 180,E1 10643.007,E2 10643.007} C_VEL
LIN {X 0,Y 329.766,Z 892.633,A -85,B 0,C 180,E1 10641.431,E2 10641.431} C_VEL
LIN {X 0,Y 339.294,Z 872.562,A -85,B 0,C 180,E1 10640.169,E2 10640.169} C_VEL
LIN {X 0,Y 348.535,Z 850.03,A -85,B 0,C 180,E1 10639.042,E2 10639.042} C_VEL
LIN {X 0,Y 355.376,Z 830.704,A -85,B 0,C 180,E1 10638.27,E2 10638.27} C_VEL
LIN {X 0,Y 362.468,Z 807.01,A -85,B 0,C 180,E1 10637.512,E2 10637.512} C_VEL
LIN {X 0,Y 367.851,Z 783.923,A -85,B 0,C 180,E1 10636.952,E2 10636.952} C_VEL
LIN {X 0,Y 372.199,Z 759.171,A -85,B 0,C 180,E1 10636.469,E2 10636.469} C_VEL
LIN {X 0,Y 377.685,Z 706.462,A -85,B 0,C 180,E1 10635.648,E2 10635.648} C_VEL
LIN {X 0,Y 388.874,Z 592.849,A -85,B 0,C 180,E1 10633.911,E2 10633.911} C_VEL
LIN {X 0,Y 385.178,Z 585.215,A -85,B 0,C 180,E1 10631.075,E2 10631.075} C_VEL
LIN {X 0,Y 382.747,Z 580.59,A -85,B 0,C 180,E1 10628.791,E2 10628.791} C_VEL
LIN {X 0,Y 381.276,Z 577.69,A -85,B 0,C 180,E1 10627.08,E2 10627.08} C_VEL
LIN {X 0,Y 379.622,Z 574.257,A -85,B 0,C 180,E1 10624.532,E2 10624.532} C_VEL
LIN {X 0,Y 378.213,Z 570.273,A -85,B 0,C 180,E1 10618.637,E2 10618.637} C_VEL
LIN {X 0,Y 379.97,Z 574.909,A -85,B 0,C 180,E1 10612.439,E2 10612.439} C_VEL
LIN {X 0,Y 382.225,Z 579.469,A -85,B 0,C 180,E1 10609.372,E2 10609.372} C_VEL
LIN {X 0,Y 384.766,Z 584.495,A -85,B 0,C 180,E1 10606.857,E2 10606.857} C_VEL
LIN {X 0,Y 388.192,Z 591.377,A -85,B 0,C 180,E1 10604.155,E2 10604.155} C_VEL
LIN {X 0,Y 388.843,Z 592.94,A -85,B 0,C 180,E1 10603.683,E2 10603.683} C_VEL
LIN {X 0,Y 373.131,Z 749.354,A -85,B 0,C 180,E1 10601.32,E2 10601.32} C_VEL
LIN {X 0,Y 368.838,Z 775.592,A -85,B 0,C 180,E1 10600.807,E2 10600.807} C_VEL
LIN {X 0,Y 364.12,Z 796.672,A -85,B 0,C 180,E1 10600.266,E2 10600.266} C_VEL
LIN {X 0,Y 357.192,Z 821.284,A -85,B 0,C 180,E1 10599.45,E2 10599.45} C_VEL
LIN {X 0,Y 349.776,Z 842.793,A -85,B 0,C 180,E1 10598.536,E2 10598.536} C_VEL
LIN {X 0,Y 340.742,Z 865.252,A -85,B 0,C 180,E1 10597.351,E2 10597.351} C_VEL
LIN {X 0,Y 331.462,Z 884.983,A -85,B 0,C 180,E1 10596.068,E2 10596.068} C_VEL
LIN {X 0,Y 321.189,Z 904.555,A -85,B 0,C 180,E1 10594.528,E2 10594.528} C_VEL
LIN {X 0,Y 309.619,Z 923.998,A -85,B 0,C 180,E1 10592.634,E2 10592.634} C_VEL
LIN {X 0,Y 298.756,Z 940.592,A -85,B 0,C 180,E1 10590.675,E2 10590.675} C_VEL
LIN {X 0,Y 285.424,Z 959.111,A -85,B 0,C 180,E1 10587.97,E2 10587.97} C_VEL
LIN {X 0,Y 274.417,Z 973.146,A -85,B 0,C 180,E1 10585.434,E2 10585.434} C_VEL
LIN {X 0,Y 261.441,Z 988.661,A -85,B 0,C 180,E1 10581.985,E2 10581.985} C_VEL
LIN {X 0,Y 249.428,Z 1001.97,A -85,B 0,C 180,E1 10578.213,E2 10578.213} C_VEL
LIN {X 0,Y 238.014,Z 1014.207,A -85,B 0,C 180,E1 10573.881,E2 10573.881} C_VEL
LIN {X 0,Y 227.439,Z 1025.012,A -85,B 0,C 180,E1 10568.908,E2 10568.908} C_VEL
LIN {X 0,Y 218.628,Z 1034.114,A -85,B 0,C 180,E1 10563.6,E2 10563.6} C_VEL
LIN {X 0,Y 210.957,Z 1042.177,A -85,B 0,C 180,E1 10557.371,E2 10557.371} C_VEL
LIN {X 0,Y 205.838,Z 1048.089,A -85,B 0,C 180,E1 10551.366,E2 10551.366} C_VEL
LIN {X 0,Y 202.099,Z 1053.164,A -85,B 0,C 180,E1 10544.136,E2 10544.136} C_VEL
LIN {X 0,Y 200.612,Z 1055.901,A -85,B 0,C 180,E1 10538.311,E2 10538.311} C_VEL
LIN {X 0,Y 200.103,Z 1057.542,A -85,B 0,C 180,E1 10532.578,E2 10532.578} C_VEL
LIN {X 0,Y 200.027,Z 1058.167,A -85,B 0,C 180,E1 10526.848,E2 10526.848} C_VEL
LIN {X 0,Y 200.279,Z 1057.583,A -85,B 0,C 180,E1 10520.807,E2 10520.807} C_VEL
LIN {X 0,Y 201.185,Z 1055.965,A -85,B 0,C 180,E1 10515.022,E2 10515.022} C_VEL
LIN {X 0,Y 203.399,Z 1053.134,A -85,B 0,C 180,E1 10508.97,E2 10508.97} C_VEL
LIN {X 0,Y 208.332,Z 1047.87,A -85,B 0,C 180,E1 10501.631,E2 10501.631} C_VEL
LIN {X 0,Y 214.24,Z 1042.154,A -85,B 0,C 180,E1 10495.94,E2 10495.94} C_VEL
LIN {X 0,Y 223.512,Z 1033.565,A -85,B 0,C 180,E1 10489.559,E2 10489.559} C_VEL
LIN {X 0,Y 233.081,Z 1024.672,A -85,B 0,C 180,E1 10484.592,E2 10484.592} C_VEL
LIN {X 0,Y 245.266,Z 1013.131,A -85,B 0,C 180,E1 10479.6,E2 10479.6} C_VEL
LIN {X 0,Y 256.9,Z 1001.514,A -85,B 0,C 180,E1 10475.72,E2 10475.72} C_VEL
LIN {X 0,Y 270.107,Z 987.682,A -85,B 0,C 180,E1 10472.036,E2 10472.036} C_VEL
LIN {X 0,Y 283.27,Z 972.632,A -85,B 0,C 180,E1 10468.908,E2 10468.908} C_VEL
LIN {X 0,Y 296.816,Z 956.045,A -85,B 0,C 180,E1 10466.134,E2 10466.134} C_VEL
LIN {X 0,Y 309.747,Z 938.391,A -85,B 0,C 180,E1 10463.798,E2 10463.798} C_VEL
LIN {X 0,Y 322.446,Z 919.477,A -85,B 0,C 180,E1 10461.763,E2 10461.763} C_VEL
LIN {X 0,Y 334.208,Z 899.531,A -85,B 0,C 180,E1 10460.044,E2 10460.044} C_VEL
LIN {X 0,Y 344.589,Z 879.973,A -85,B 0,C 180,E1 10458.666,E2 10458.666} C_VEL
LIN {X 0,Y 354.703,Z 857.899,A -85,B 0,C 180,E1 10457.405,E2 10457.405} C_VEL
LIN {X 0,Y 362.288,Z 838.902,A -85,B 0,C 180,E1 10456.516,E2 10456.516} C_VEL
LIN {X 0,Y 370.59,Z 814.284,A -85,B 0,C 180,E1 10455.587,E2 10455.587} C_VEL
LIN {X 0,Y 376.482,Z 792.686,A -85,B 0,C 180,E1 10454.949,E2 10454.949} C_VEL
LIN {X 0,Y 381.881,Z 767.46,A -85,B 0,C 180,E1 10454.381,E2 10454.381} C_VEL
LIN {X 0,Y 385.279,Z 744.593,A -85,B 0,C 180,E1 10453.991,E2 10453.991} C_VEL
LIN {X 0,Y 399.969,Z 601.459,A -85,B 0,C 180,E1 10451.869,E2 10451.869} C_VEL
LIN {X 0,Y 396.863,Z 595.024,A -85,B 0,C 180,E1 10449.06,E2 10449.06} C_VEL
LIN {X 0,Y 395.065,Z 591.422,A -85,B 0,C 180,E1 10446.978,E2 10446.978} C_VEL
LIN {X 0,Y 393.517,Z 588.118,A -85,B 0,C 180,E1 10444.518,E2 10444.518} C_VEL
LIN {X 0,Y 392.243,Z 584.508,A -85,B 0,C 180,E1 10438.978,E2 10438.978} C_VEL
LIN {X 0,Y 393.803,Z 588.669,A -85,B 0,C 180,E1 10433.293,E2 10433.293} C_VEL
LIN {X 0,Y 394.497,Z 590.432,A -85,B 0,C 180,E1 10432.124,E2 10432.124} C_VEL
LIN {X 0,Y 394.865,Z 592.475,A -85,B 0,C 180,E1 10431.429,E2 10431.429} C_VEL
LIN {X 0,Y 395.442,Z 601.545,A -85,B 0,C 180,E1 10429.792,E2 10429.792} C_VEL
LIN {X 0,Y 395.919,Z 603.34,A -85,B 0,C 180,E1 10429.197,E2 10429.197} C_VEL
LIN {X 0,Y 397.764,Z 607.479,A -85,B 0,C 180,E1 10427.423,E2 10427.423} C_VEL
LIN {X 0,Y 382.227,Z 754.858,A -85,B 0,C 180,E1 10425.29,E2 10425.29} C_VEL
LIN {X 0,Y 377.68,Z 781.364,A -85,B 0,C 180,E1 10424.826,E2 10424.826} C_VEL
LIN {X 0,Y 372.538,Z 803.082,A -85,B 0,C 180,E1 10424.363,E2 10424.363} C_VEL
LIN {X 0,Y 365.168,Z 827.678,A -85,B 0,C 180,E1 10423.684,E2 10423.684} C_VEL
LIN {X 0,Y 357.68,Z 848.26,A -85,B 0,C 180,E1 10422.952,E2 10422.952} C_VEL
LIN {X 0,Y 348.118,Z 870.897,A -85,B 0,C 180,E1 10421.938,E2 10421.938} C_VEL
LIN {X 0,Y 338.26,Z 890.87,A -85,B 0,C 180,E1 10420.81,E2 10420.81} C_VEL
LIN {X 0,Y 327.717,Z 909.962,A -85,B 0,C 180,E1 10419.501,E2 10419.501} C_VEL
LIN {X 0,Y 314.908,Z 930.438,A -85,B 0,C 180,E1 10417.754,E2 10417.754} C_VEL
LIN {X 0,Y 303.245,Z 947.288,A -85,B 0,C 180,E1 10415.973,E2 10415.973} C_VEL
LIN {X 0,Y 288.462,Z 966.61,A -85,B 0,C 180,E1 10413.419,E2 10413.419} C_VEL
LIN {X 0,Y 275.782,Z 981.731,A -85,B 0,C 180,E1 10410.901,E2 10410.901} C_VEL
LIN {X 0,Y 260.951,Z 998.085,A -85,B 0,C 180,E1 10407.456,E2 10407.456} C_VEL
LIN {X 0,Y 248.428,Z 1010.917,A -85,B 0,C 180,E1 10403.998,E2 10403.998} C_VEL
LIN {X 0,Y 235.162,Z 1023.861,A -85,B 0,C 180,E1 10399.561,E2 10399.561} C_VEL
LIN {X 0,Y 223.908,Z 1034.335,A -85,B 0,C 180,E1 10394.876,E2 10394.876} C_VEL
LIN {X 0,Y 213.377,Z 1044.148,A -85,B 0,C 180,E1 10389.243,E2 10389.243} C_VEL
LIN {X 0,Y 204.895,Z 1052.03,A -85,B 0,C 180,E1 10383.131,E2 10383.131} C_VEL
LIN {X 0,Y 198.394,Z 1058.688,A -85,B 0,C 180,E1 10376.328,E2 10376.328} C_VEL
LIN {X 0,Y 194.289,Z 1063.487,A -85,B 0,C 180,E1 10369.231,E2 10369.231} C_VEL
LIN {X 0,Y 192.492,Z 1066.42,A -85,B 0,C 180,E1 10362.907,E2 10362.907} C_VEL
LIN {X 0,Y 191.983,Z 1068.226,A -85,B 0,C 180,E1 10356.279,E2 10356.279} C_VEL
LIN {X 0,Y 192.028,Z 1068.581,A -85,B 0,C 180,E1 10350.597,E2 10350.597} C_VEL
LIN {X 0,Y 191.992,Z 1067.983,A -85,B 0,C 180,E1 10345.22,E2 10345.22} C_VEL
LIN {X 0,Y 192.171,Z 1066.342,A -85,B 0,C 180,E1 10339.507,E2 10339.507} C_VEL
LIN {X 0,Y 193.206,Z 1063.684,A -85,B 0,C 180,E1 10333.772,E2 10333.772} C_VEL
LIN {X 0,Y 196.132,Z 1059.144,A -85,B 0,C 180,E1 10326.887,E2 10326.887} C_VEL
LIN {X 0,Y 201.435,Z 1052.554,A -85,B 0,C 180,E1 10319.911,E2 10319.911} C_VEL
LIN {X 0,Y 208.411,Z 1045.038,A -85,B 0,C 180,E1 10313.835,E2 10313.835} C_VEL
LIN {X 0,Y 217.789,Z 1035.358,A -85,B 0,C 180,E1 10307.91,E2 10307.91} C_VEL
LIN {X 0,Y 227.563,Z 1025.418,A -85,B 0,C 180,E1 10303.165,E2 10303.165} C_VEL
LIN {X 0,Y 240.456,Z 1012.008,A -85,B 0,C 180,E1 10298.194,E2 10298.194} C_VEL
LIN {X 0,Y 251.991,Z 999.478,A -85,B 0,C 180,E1 10294.571,E2 10294.571} C_VEL
LIN {X 0,Y 265.797,Z 983.634,A -85,B 0,C 180,E1 10290.94,E2 10290.94} C_VEL
LIN {X 0,Y 277.981,Z 968.517,A -85,B 0,C 180,E1 10288.206,E2 10288.206} C_VEL
LIN {X 0,Y 291.141,Z 950.998,A -85,B 0,C 180,E1 10285.641,E2 10285.641} C_VEL
LIN {X 0,Y 303.234,Z 933.066,A -85,B 0,C 180,E1 10283.554,E2 10283.554} C_VEL
LIN {X 0,Y 314.492,Z 914.848,A -85,B 0,C 180,E1 10281.816,E2 10281.816} C_VEL
LIN {X 0,Y 326.04,Z 893.828,A -85,B 0,C 180,E1 10280.21,E2 10280.21} C_VEL
LIN {X 0,Y 335.282,Z 874.861,A -85,B 0,C 180,E1 10279.027,E2 10279.027} C_VEL
LIN {X 0,Y 345.114,Z 851.78,A -85,B 0,C 180,E1 10277.87,E2 10277.87} C_VEL
LIN {X 0,Y 352.486,Z 831.425,A -85,B 0,C 180,E1 10277.068,E2 10277.068} C_VEL
LIN {X 0,Y 359.498,Z 808.699,A -85,B 0,C 180,E1 10276.349,E2 10276.349} C_VEL
LIN {X 0,Y 365.249,Z 784.701,A -85,B 0,C 180,E1 10275.775,E2 10275.775} C_VEL
LIN {X 0,Y 369.558,Z 761.001,A -85,B 0,C 180,E1 10275.318,E2 10275.318} C_VEL
LIN {X 0,Y 373.795,Z 722.938,A -85,B 0,C 180,E1 10274.723,E2 10274.723} C_VEL
LIN {X 0,Y 386.335,Z 598.311,A -85,B 0,C 180,E1 10272.861,E2 10272.861} C_VEL
LIN {X 0,Y 383.013,Z 591.33,A -85,B 0,C 180,E1 10270.073,E2 10270.073} C_VEL
LIN {X 0,Y 380.415,Z 585.945,A -85,B 0,C 180,E1 10267.248,E2 10267.248} C_VEL
LIN {X 0,Y 378.474,Z 582.039,A -85,B 0,C 180,E1 10264.242,E2 10264.242} C_VEL
LIN {X 0,Y 377.231,Z 578.267,A -85,B 0,C 180,E1 10258.633,E2 10258.633} C_VEL
LIN {X 0,Y 378.855,Z 582.72,A -85,B 0,C 180,E1 10252.646,E2 10252.646} C_VEL
LIN {X 0,Y 380.974,Z 587.166,A -85,B 0,C 180,E1 10249.643,E2 10249.643} C_VEL
LIN {X 0,Y 383.435,Z 592.202,A -85,B 0,C 180,E1 10247.117,E2 10247.117} C_VEL
LIN {X 0,Y 386.293,Z 598.234,A -85,B 0,C 180,E1 10244.753,E2 10244.753} C_VEL
LIN {X 0,Y 370.781,Z 749.609,A -85,B 0,C 180,E1 10242.498,E2 10242.498} C_VEL
LIN {X 0,Y 366.405,Z 775.895,A -85,B 0,C 180,E1 10241.995,E2 10241.995} C_VEL
LIN {X 0,Y 361.614,Z 796.958,A -85,B 0,C 180,E1 10241.468,E2 10241.468} C_VEL
LIN {X 0,Y 354.469,Z 821.873,A -85,B 0,C 180,E1 10240.658,E2 10240.658} C_VEL
LIN {X 0,Y 347.304,Z 842.342,A -85,B 0,C 180,E1 10239.81,E2 10239.81} C_VEL
LIN {X 0,Y 338.154,Z 864.84,A -85,B 0,C 180,E1 10238.658,E2 10238.658} C_VEL
LIN {X 0,Y 328.289,Z 885.437,A -85,B 0,C 180,E1 10237.349,E2 10237.349} C_VEL
LIN {X 0,Y 317.416,Z 905.713,A -85,B 0,C 180,E1 10235.777,E2 10235.777} C_VEL
LIN {X 0,Y 305.607,Z 924.995,A -85,B 0,C 180,E1 10233.911,E2 10233.911} C_VEL
LIN {X 0,Y 294.254,Z 941.888,A -85,B 0,C 180,E1 10231.928,E2 10231.928} C_VEL
LIN {X 0,Y 281.209,Z 959.465,A -85,B 0,C 180,E1 10229.37,E2 10229.37} C_VEL
LIN {X 0,Y 269.204,Z 974.323,A -85,B 0,C 180,E1 10226.689,E2 10226.689} C_VEL
LIN {X 0,Y 255.218,Z 990.363,A -85,B 0,C 180,E1 10223.057,E2 10223.057} C_VEL
LIN {X 0,Y 243.481,Z 1002.907,A -85,B 0,C 180,E1 10219.44,E2 10219.44} C_VEL
LIN {X 0,Y 230.949,Z 1015.708,A -85,B 0,C 180,E1 10214.762,E2 10214.762} C_VEL
LIN {X 0,Y 220.75,Z 1025.688,A -85,B 0,C 180,E1 10210.03,E2 10210.03} C_VEL
LIN {X 0,Y 211.127,Z 1035.168,A -85,B 0,C 180,E1 10204.304,E2 10204.304} C_VEL
LIN {X 0,Y 203.473,Z 1042.736,A -85,B 0,C 180,E1 10198.148,E2 10198.148} C_VEL
LIN {X 0,Y 197.87,Z 1048.88,A -85,B 0,C 180,E1 10191.595,E2 10191.595} C_VEL
LIN {X 0,Y 194.225,Z 1053.482,A -85,B 0,C 180,E1 10184.568,E2 10184.568} C_VEL
LIN {X 0,Y 192.665,Z 1056.132,A -85,B 0,C 180,E1 10178.656,E2 10178.656} C_VEL
LIN {X 0,Y 192.109,Z 1057.766,A -85,B 0,C 180,E1 10172.685,E2 10172.685} C_VEL
LIN {X 0,Y 192.031,Z 1058.383,A -85,B 0,C 180,E1 10166.716,E2 10166.716} C_VEL
LIN {X 0,Y 192.288,Z 1057.854,A -85,B 0,C 180,E1 10160.723,E2 10160.723} C_VEL
LIN {X 0,Y 193.332,Z 1056.165,A -85,B 0,C 180,E1 10154.399,E2 10154.399} C_VEL
LIN {X 0,Y 195.766,Z 1053.328,A -85,B 0,C 180,E1 10148.108,E2 10148.108} C_VEL
LIN {X 0,Y 201.105,Z 1048.051,A -85,B 0,C 180,E1 10140.513,E2 10140.513} C_VEL
LIN {X 0,Y 207.429,Z 1042.328,A -85,B 0,C 180,E1 10134.659,E2 10134.659} C_VEL
LIN {X 0,Y 217.266,Z 1033.724,A -85,B 0,C 180,E1 10128.14,E2 10128.14} C_VEL
LIN {X 0,Y 227.331,Z 1024.823,A -85,B 0,C 180,E1 10123.102,E2 10123.102} C_VEL
LIN {X 0,Y 240.184,Z 1013.15,A -85,B 0,C 180,E1 10118.034,E2 10118.034} C_VEL
LIN {X 0,Y 252.413,Z 1001.383,A -85,B 0,C 180,E1 10114.115,E2 10114.115} C_VEL
LIN {X 0,Y 265.872,Z 987.724,A -85,B 0,C 180,E1 10110.511,E2 10110.511} C_VEL
LIN {X 0,Y 279.379,Z 972.724,A -85,B 0,C 180,E1 10107.428,E2 10107.428} C_VEL
LIN {X 0,Y 293.373,Z 956.006,A -85,B 0,C 180,E1 10104.678,E2 10104.678} C_VEL
LIN {X 0,Y 306.579,Z 938.377,A -85,B 0,C 180,E1 10102.389,E2 10102.389} C_VEL
LIN {X 0,Y 319.51,Z 919.5,A -85,B 0,C 180,E1 10100.402,E2 10100.402} C_VEL
LIN {X 0,Y 331.503,Z 899.528,A -85,B 0,C 180,E1 10098.72,E2 10098.72} C_VEL
LIN {X 0,Y 342.502,Z 879.137,A -85,B 0,C 180,E1 10097.324,E2 10097.324} C_VEL
LIN {X 0,Y 352.348,Z 857.848,A -85,B 0,C 180,E1 10096.147,E2 10096.147} C_VEL
LIN {X 0,Y 360.134,Z 838.623,A -85,B 0,C 180,E1 10095.275,E2 10095.275} C_VEL
LIN {X 0,Y 368.502,Z 814.062,A -85,B 0,C 180,E1 10094.378,E2 10094.378} C_VEL
LIN {X 0,Y 374.417,Z 792.649,A -85,B 0,C 180,E1 10093.763,E2 10093.763} C_VEL
LIN {X 0,Y 379.943,Z 766.994,A -85,B 0,C 180,E1 10093.204,E2 10093.204} C_VEL
LIN {X 0,Y 383.325,Z 744.44,A -85,B 0,C 180,E1 10092.83,E2 10092.83} C_VEL
LIN {X 0,Y 397.689,Z 607.171,A -85,B 0,C 180,E1 10090.833,E2 10090.833} C_VEL
LIN {X 0,Y 395.192,Z 601.942,A -85,B 0,C 180,E1 10088.365,E2 10088.365} C_VEL
LIN {X 0,Y 393.858,Z 599.124,A -85,B 0,C 180,E1 10086.706,E2 10086.706} C_VEL
LIN {X 0,Y 392.459,Z 596,A -85,B 0,C 180,E1 10084.384,E2 10084.384} C_VEL
LIN {X 0,Y 391.263,Z 592.483,A -85,B 0,C 180,E1 10078.975,E2 10078.975} C_VEL
LIN {X 0,Y 392.699,Z 596.479,A -85,B 0,C 180,E1 10073.494,E2 10073.494} C_VEL
LIN {X 0,Y 394.717,Z 600.935,A -85,B 0,C 180,E1 10070.523,E2 10070.523} C_VEL
LIN {X 0,Y 395.919,Z 603.34,A -85,B 0,C 180,E1 10069.197,E2 10069.197} C_VEL
LIN {X 0,Y 396.183,Z 604.959,A -85,B 0,C 180,E1 10068.822,E2 10068.822} C_VEL
LIN {X 0,Y 396.148,Z 608.307,A -85,B 0,C 180,E1 10068.524,E2 10068.524} C_VEL
LIN {X 0,Y 395.721,Z 613.49,A -85,B 0,C 180,E1 10068.355,E2 10068.355} C_VEL
LIN {X 0,Y 394.184,Z 626.449,A -85,B 0,C 180,E1 10068.292,E2 10068.292} C_VEL
LIN {X 0,Y 380.379,Z 754.832,A -85,B 0,C 180,E1 10066.463,E2 10066.463} C_VEL
LIN {X 0,Y 375.788,Z 781.17,A -85,B 0,C 180,E1 10066.014,E2 10066.014} C_VEL
LIN {X 0,Y 370.573,Z 802.913,A -85,B 0,C 180,E1 10065.565,E2 10065.565} C_VEL
LIN {X 0,Y 362.861,Z 828.205,A -85,B 0,C 180,E1 10064.887,E2 10064.887} C_VEL
LIN {X 0,Y 355.143,Z 849.027,A -85,B 0,C 180,E1 10064.165,E2 10064.165} C_VEL
LIN {X 0,Y 344.823,Z 872.731,A -85,B 0,C 180,E1 10063.118,E2 10063.118} C_VEL
LIN {X 0,Y 334.825,Z 892.502,A -85,B 0,C 180,E1 10062.015,E2 10062.015} C_VEL
LIN {X 0,Y 322.843,Z 913.487,A -85,B 0,C 180,E1 10060.575,E2 10060.575} C_VEL
LIN {X 0,Y 310.673,Z 932.218,A -85,B 0,C 180,E1 10058.964,E2 10058.964} C_VEL
LIN {X 0,Y 297.194,Z 951.1,A -85,B 0,C 180,E1 10056.951,E2 10056.951} C_VEL
LIN {X 0,Y 283.332,Z 968.379,A -85,B 0,C 180,E1 10054.613,E2 10054.613} C_VEL
LIN {X 0,Y 268.909,Z 985.024,A -85,B 0,C 180,E1 10051.792,E2 10051.792} C_VEL
LIN {X 0,Y 254.505,Z 1000.079,A -85,B 0,C 180,E1 10048.489,E2 10048.489} C_VEL
LIN {X 0,Y 240.984,Z 1013.417,A -85,B 0,C 180,E1 10044.778,E2 10044.778} C_VEL
LIN {X 0,Y 227.523,Z 1025.793,A -85,B 0,C 180,E1 10040.27,E2 10040.27} C_VEL
LIN {X 0,Y 216.047,Z 1036.037,A -85,B 0,C 180,E1 10035.457,E2 10035.457} C_VEL
LIN {X 0,Y 204.88,Z 1045.773,A -85,B 0,C 180,E1 10029.379,E2 10029.379} C_VEL
LIN {X 0,Y 197.008,Z 1052.779,A -85,B 0,C 180,E1 10023.588,E2 10023.588} C_VEL
LIN {X 0,Y 189.904,Z 1059.588,A -85,B 0,C 180,E1 10015.914,E2 10015.914} C_VEL
LIN {X 0,Y 186.313,Z 1063.62,A -85,B 0,C 180,E1 10009.435,E2 10009.435} C_VEL
LIN {X 0,Y 184.372,Z 1066.692,A -85,B 0,C 180,E1 10002.211,E2 10002.211} C_VEL
LIN {X 0,Y 183.987,Z 1068.12,A -85,B 0,C 180,E1 9995.301,E2 9995.301} C_VEL
LIN {X 0,Y 184.042,Z 1068.32,A -85,B 0,C 180,E1 9990,E2 9990} C_VEL
LIN {X 0,Y 183.994,Z 1067.689,A -85,B 0,C 180,E1 9984.699,E2 9984.699} C_VEL
LIN {X 0,Y 184.213,Z 1066.11,A -85,B 0,C 180,E1 9979.049,E2 9979.049} C_VEL
LIN {X 0,Y 185.383,Z 1063.444,A -85,B 0,C 180,E1 9973.067,E2 9973.067} C_VEL
LIN {X 0,Y 188.729,Z 1058.733,A -85,B 0,C 180,E1 9965.681,E2 9965.681} C_VEL
LIN {X 0,Y 194.349,Z 1052.257,A -85,B 0,C 180,E1 9958.654,E2 9958.654} C_VEL
LIN {X 0,Y 201.777,Z 1044.768,A -85,B 0,C 180,E1 9952.445,E2 9952.445} C_VEL
LIN {X 0,Y 211.697,Z 1035.072,A -85,B 0,C 180,E1 9946.403,E2 9946.403} C_VEL
LIN {X 0,Y 221.962,Z 1025.124,A -85,B 0,C 180,E1 9941.6,E2 9941.6} C_VEL
LIN {X 0,Y 235.414,Z 1011.697,A -85,B 0,C 180,E1 9936.606,E2 9936.606} C_VEL
LIN {X 0,Y 247.035,Z 999.528,A -85,B 0,C 180,E1 9933.087,E2 9933.087} C_VEL
LIN {X 0,Y 260.925,Z 984.152,A -85,B 0,C 180,E1 9929.555,E2 9929.555} C_VEL
LIN {X 0,Y 273.425,Z 969.105,A -85,B 0,C 180,E1 9926.838,E2 9926.838} C_VEL
LIN {X 0,Y 286.498,Z 952.213,A -85,B 0,C 180,E1 9924.37,E2 9924.37} C_VEL
LIN {X 0,Y 299.686,Z 933.231,A -85,B 0,C 180,E1 9922.175,E2 9922.175} C_VEL
LIN {X 0,Y 311.129,Z 915.119,A -85,B 0,C 180,E1 9920.478,E2 9920.478} C_VEL
LIN {X 0,Y 323.314,Z 893.384,A -85,B 0,C 180,E1 9918.854,E2 9918.854} C_VEL
LIN {X 0,Y 332.718,Z 874.391,A -85,B 0,C 180,E1 9917.702,E2 9917.702} C_VEL
LIN {X 0,Y 343.146,Z 850.106,A -85,B 0,C 180,E1 9916.53,E2 9916.53} C_VEL
LIN {X 0,Y 350.637,Z 829.556,A -85,B 0,C 180,E1 9915.756,E2 9915.756} C_VEL
LIN {X 0,Y 358.046,Z 805.186,A -85,B 0,C 180,E1 9915.034,E2 9915.034} C_VEL
LIN {X 0,Y 363.333,Z 782.986,A -85,B 0,C 180,E1 9914.531,E2 9914.531} C_VEL
LIN {X 0,Y 367.777,Z 758.119,A -85,B 0,C 180,E1 9914.071,E2 9914.071} C_VEL
LIN {X 0,Y 373.825,Z 701.889,A -85,B 0,C 180,E1 9913.224,E2 9913.224} C_VEL
LIN {X 0,Y 383.88,Z 603.704,A -85,B 0,C 180,E1 9911.76,E2 9911.76} C_VEL
LIN {X 0,Y 380.828,Z 597.123,A -85,B 0,C 180,E1 9908.912,E2 9908.912} C_VEL
LIN {X 0,Y 378.954,Z 593.28,A -85,B 0,C 180,E1 9906.667,E2 9906.667} C_VEL
LIN {X 0,Y 377.415,Z 589.918,A -85,B 0,C 180,E1 9904.102,E2 9904.102} C_VEL
LIN {X 0,Y 376.262,Z 586.148,A -85,B 0,C 180,E1 9898.782,E2 9898.782} C_VEL
LIN {X 0,Y 377.784,Z 590.646,A -85,B 0,C 180,E1 9892.778,E2 9892.778} C_VEL
LIN {X 0,Y 379.731,Z 594.863,A -85,B 0,C 180,E1 9889.915,E2 9889.915} C_VEL
LIN {X 0,Y 382.439,Z 600.521,A -85,B 0,C 180,E1 9887.083,E2 9887.083} C_VEL
LIN {X 0,Y 383.853,Z 603.775,A -85,B 0,C 180,E1 9885.834,E2 9885.834} C_VEL
LIN {X 0,Y 368.589,Z 749.865,A -85,B 0,C 180,E1 9883.691,E2 9883.691} C_VEL
LIN {X 0,Y 364.159,Z 776.069,A -85,B 0,C 180,E1 9883.201,E2 9883.201} C_VEL
LIN {X 0,Y 359.246,Z 797.335,A -85,B 0,C 180,E1 9882.683,E2 9882.683} C_VEL
LIN {X 0,Y 351.905,Z 822.461,A -85,B 0,C 180,E1 9881.885,E2 9881.885} C_VEL
LIN {X 0,Y 344.628,Z 842.885,A -85,B 0,C 180,E1 9881.057,E2 9881.057} C_VEL
LIN {X 0,Y 335.322,Z 865.317,A -85,B 0,C 180,E1 9879.933,E2 9879.933} C_VEL
LIN {X 0,Y 325.283,Z 885.89,A -85,B 0,C 180,E1 9878.653,E2 9878.653} C_VEL
LIN {X 0,Y 314.2,Z 906.14,A -85,B 0,C 180,E1 9877.115,E2 9877.115} C_VEL
LIN {X 0,Y 302.146,Z 925.391,A -85,B 0,C 180,E1 9875.285,E2 9875.285} C_VEL
LIN {X 0,Y 290.027,Z 942.998,A -85,B 0,C 180,E1 9873.243,E2 9873.243} C_VEL
LIN {X 0,Y 276.426,Z 960.733,A -85,B 0,C 180,E1 9870.662,E2 9870.662} C_VEL
LIN {X 0,Y 264.126,Z 975.499,A -85,B 0,C 180,E1 9867.993,E2 9867.993} C_VEL
LIN {X 0,Y 249.749,Z 991.375,A -85,B 0,C 180,E1 9864.363,E2 9864.363} C_VEL
LIN {X 0,Y 238.266,Z 1003.221,A -85,B 0,C 180,E1 9860.928,E2 9860.928} C_VEL
LIN {X 0,Y 225.426,Z 1015.823,A -85,B 0,C 180,E1 9856.302,E2 9856.302} C_VEL
LIN {X 0,Y 214.568,Z 1025.975,A -85,B 0,C 180,E1 9851.431,E2 9851.431} C_VEL
LIN {X 0,Y 204.441,Z 1035.44,A -85,B 0,C 180,E1 9845.592,E2 9845.592} C_VEL
LIN {X 0,Y 196.331,Z 1042.999,A -85,B 0,C 180,E1 9839.269,E2 9839.269} C_VEL
LIN {X 0,Y 190.381,Z 1049.094,A -85,B 0,C 180,E1 9832.544,E2 9832.544} C_VEL
LIN {X 0,Y 186.436,Z 1053.7,A -85,B 0,C 180,E1 9825.236,E2 9825.236} C_VEL
LIN {X 0,Y 184.724,Z 1056.364,A -85,B 0,C 180,E1 9819.031,E2 9819.031} C_VEL
LIN {X 0,Y 184.116,Z 1057.99,A -85,B 0,C 180,E1 9812.801,E2 9812.801} C_VEL
LIN {X 0,Y 184.031,Z 1058.577,A -85,B 0,C 180,E1 9806.885,E2 9806.885} C_VEL
LIN {X 0,Y 184.297,Z 1058.124,A -85,B 0,C 180,E1 9800.633,E2 9800.633} C_VEL
LIN {X 0,Y 185.411,Z 1056.475,A -85,B 0,C 180,E1 9794.036,E2 9794.036} C_VEL
LIN {X 0,Y 187.847,Z 1053.833,A -85,B 0,C 180,E1 9787.795,E2 9787.795} C_VEL
LIN {X 0,Y 192.889,Z 1049.228,A -85,B 0,C 180,E1 9780.498,E2 9780.498} C_VEL
LIN {X 0,Y 200.005,Z 1043.098,A -85,B 0,C 180,E1 9773.849,E2 9773.849} C_VEL
LIN {X 0,Y 209.332,Z 1035.472,A -85,B 0,C 180,E1 9767.662,E2 9767.662} C_VEL
LIN {X 0,Y 220.668,Z 1025.882,A -85,B 0,C 180,E1 9762.002,E2 9762.002} C_VEL
LIN {X 0,Y 233.222,Z 1015.086,A -85,B 0,C 180,E1 9757.114,E2 9757.114} C_VEL
LIN {X 0,Y 246.535,Z 1002.768,A -85,B 0,C 180,E1 9752.908,E2 9752.908} C_VEL
LIN {X 0,Y 259.579,Z 990.037,A -85,B 0,C 180,E1 9749.478,E2 9749.478} C_VEL
LIN {X 0,Y 274.176,Z 974.5,A -85,B 0,C 180,E1 9746.216,E2 9746.216} C_VEL
LIN {X 0,Y 286.421,Z 960.373,A -85,B 0,C 180,E1 9743.846,E2 9743.846} C_VEL
LIN {X 0,Y 301.525,Z 941.2,A -85,B 0,C 180,E1 9741.279,E2 9741.279} C_VEL
LIN {X 0,Y 313.493,Z 924.303,A -85,B 0,C 180,E1 9739.475,E2 9739.475} C_VEL
LIN {X 0,Y 326.855,Z 903.201,A -85,B 0,C 180,E1 9737.651,E2 9737.651} C_VEL
LIN {X 0,Y 337.283,Z 884.528,A -85,B 0,C 180,E1 9736.358,E2 9736.358} C_VEL
LIN {X 0,Y 348.01,Z 862.771,A -85,B 0,C 180,E1 9735.12,E2 9735.12} C_VEL
LIN {X 0,Y 356.801,Z 841.79,A -85,B 0,C 180,E1 9734.159,E2 9734.159} C_VEL
LIN {X 0,Y 364.795,Z 819.642,A -85,B 0,C 180,E1 9733.334,E2 9733.334} C_VEL
LIN {X 0,Y 371.694,Z 795.793,A -85,B 0,C 180,E1 9732.645,E2 9732.645} C_VEL
LIN {X 0,Y 376.98,Z 772.958,A -85,B 0,C 180,E1 9732.137,E2 9732.137} C_VEL
LIN {X 0,Y 381.079,Z 747.849,A -85,B 0,C 180,E1 9731.711,E2 9731.711} C_VEL
LIN {X 0,Y 395.525,Z 613.102,A -85,B 0,C 180,E1 9729.792,E2 9729.792} C_VEL
LIN {X 0,Y 393.149,Z 607.705,A -85,B 0,C 180,E1 9727.086,E2 9727.086} C_VEL
LIN {X 0,Y 391.328,Z 603.79,A -85,B 0,C 180,E1 9724.103,E2 9724.103} C_VEL
LIN {X 0,Y 390.283,Z 600.464,A -85,B 0,C 180,E1 9718.972,E2 9718.972} C_VEL
LIN {X 0,Y 391.634,Z 604.404,A -85,B 0,C 180,E1 9713.624,E2 9713.624} C_VEL
LIN {X 0,Y 393.488,Z 608.629,A -85,B 0,C 180,E1 9710.788,E2 9710.788} C_VEL
LIN {X 0,Y 395.592,Z 613.189,A -85,B 0,C 180,E1 9708.482,E2 9708.482} C_VEL
LIN {X 0,Y 394.184,Z 626.449,A -85,B 0,C 180,E1 9708.292,E2 9708.292} C_VEL
LIN {X 0,Y 393.172,Z 634.147,A -85,B 0,C 180,E1 9708.33,E2 9708.33} C_VEL
LIN {X 0,Y 389.82,Z 654.704,A -85,B 0,C 180,E1 9708.946,E2 9708.946} C_VEL
LIN {X 0,Y 388.977,Z 661.307,A -85,B 0,C 180,E1 9708.962,E2 9708.962} C_VEL
LIN {X 0,Y 378.64,Z 755.206,A -85,B 0,C 180,E1 9707.641,E2 9707.641} C_VEL
LIN {X 0,Y 374.022,Z 781.147,A -85,B 0,C 180,E1 9707.21,E2 9707.21} C_VEL
LIN {X 0,Y 368.738,Z 802.884,A -85,B 0,C 180,E1 9706.776,E2 9706.776} C_VEL
LIN {X 0,Y 360.827,Z 828.417,A -85,B 0,C 180,E1 9706.115,E2 9706.115} C_VEL
LIN {X 0,Y 352.851,Z 849.587,A -85,B 0,C 180,E1 9705.403,E2 9705.403} C_VEL
LIN {X 0,Y 342.123,Z 873.665,A -85,B 0,C 180,E1 9704.365,E2 9704.365} C_VEL
LIN {X 0,Y 332.417,Z 892.512,A -85,B 0,C 180,E1 9703.341,E2 9703.341} C_VEL
LIN {X 0,Y 320.236,Z 913.457,A -85,B 0,C 180,E1 9701.944,E2 9701.944} C_VEL
LIN {X 0,Y 308.266,Z 931.562,A -85,B 0,C 180,E1 9700.436,E2 9700.436} C_VEL
LIN {X 0,Y 295.322,Z 949.387,A -85,B 0,C 180,E1 9698.604,E2 9698.604} C_VEL
LIN {X 0,Y 280.673,Z 967.403,A -85,B 0,C 180,E1 9696.262,E2 9696.262} C_VEL
LIN {X 0,Y 267.373,Z 982.413,A -85,B 0,C 180,E1 9693.814,E2 9693.814} C_VEL
LIN {X 0,Y 251.736,Z 998.546,A -85,B 0,C 180,E1 9690.443,E2 9690.443} C_VEL
LIN {X 0,Y 239.086,Z 1010.653,A -85,B 0,C 180,E1 9687.204,E2 9687.204} C_VEL
LIN {X 0,Y 224.157,Z 1024.084,A -85,B 0,C 180,E1 9682.561,E2 9682.561} C_VEL
LIN {X 0,Y 211.935,Z 1034.486,A -85,B 0,C 180,E1 9677.792,E2 9677.792} C_VEL
LIN {X 0,Y 199.895,Z 1044.523,A -85,B 0,C 180,E1 9671.704,E2 9671.704} C_VEL
LIN {X 0,Y 190.89,Z 1051.982,A -85,B 0,C 180,E1 9665.551,E2 9665.551} C_VEL
LIN {X 0,Y 183.512,Z 1058.546,A -85,B 0,C 180,E1 9658.296,E2 9658.296} C_VEL
LIN {X 0,Y 178.898,Z 1063.093,A -85,B 0,C 180,E1 9650.959,E2 9650.959} C_VEL
LIN {X 0,Y 176.682,Z 1066.017,A -85,B 0,C 180,E1 9644.084,E2 9644.084} C_VEL
LIN {X 0,Y 175.988,Z 1067.831,A -85,B 0,C 180,E1 9636.525,E2 9636.525} C_VEL
LIN {X 0,Y 176.033,Z 1068.148,A -85,B 0,C 180,E1 9630.651,E2 9630.651} C_VEL
LIN {X 0,Y 175.995,Z 1067.606,A -85,B 0,C 180,E1 9625.111,E2 9625.111} C_VEL
LIN {X 0,Y 176.226,Z 1065.996,A -85,B 0,C 180,E1 9618.877,E2 9618.877} C_VEL
LIN {X 0,Y 177.583,Z 1063.204,A -85,B 0,C 180,E1 9612.299,E2 9612.299} C_VEL
LIN {X 0,Y 181.31,Z 1058.414,A -85,B 0,C 180,E1 9604.523,E2 9604.523} C_VEL
LIN {X 0,Y 187.293,Z 1052.029,A -85,B 0,C 180,E1 9597.371,E2 9597.371} C_VEL
LIN {X 0,Y 195.674,Z 1044.135,A -85,B 0,C 180,E1 9590.681,E2 9590.681} C_VEL
LIN {X 0,Y 206.266,Z 1034.318,A -85,B 0,C 180,E1 9584.554,E2 9584.554} C_VEL
LIN {X 0,Y 217.687,Z 1023.781,A -85,B 0,C 180,E1 9579.497,E2 9579.497} C_VEL
LIN {X 0,Y 231.209,Z 1010.74,A -85,B 0,C 180,E1 9574.747,E2 9574.747} C_VEL
LIN {X 0,Y 243.963,Z 997.829,A -85,B 0,C 180,E1 9571.092,E2 9571.092} C_VEL
LIN {X 0,Y 258.429,Z 982.098,A -85,B 0,C 180,E1 9567.622,E2 9567.622} C_VEL
LIN {X 0,Y 270.577,Z 967.817,A -85,B 0,C 180,E1 9565.127,E2 9565.127} C_VEL
LIN {X 0,Y 284.412,Z 950.248,A -85,B 0,C 180,E1 9562.653,E2 9562.653} C_VEL
LIN {X 0,Y 297.06,Z 932.287,A -85,B 0,C 180,E1 9560.653,E2 9560.653} C_VEL
LIN {X 0,Y 309.095,Z 913.555,A -85,B 0,C 180,E1 9558.96,E2 9558.96} C_VEL
LIN {X 0,Y 320.773,Z 892.939,A -85,B 0,C 180,E1 9557.476,E2 9557.476} C_VEL
LIN {X 0,Y 330.464,Z 873.657,A -85,B 0,C 180,E1 9556.343,E2 9556.343} C_VEL
LIN {X 0,Y 340.926,Z 849.574,A -85,B 0,C 180,E1 9555.223,E2 9555.223} C_VEL
LIN {X 0,Y 348.526,Z 828.98,A -85,B 0,C 180,E1 9554.475,E2 9554.475} C_VEL
LIN {X 0,Y 356.163,Z 803.996,A -85,B 0,C 180,E1 9553.767,E2 9553.767} C_VEL
LIN {X 0,Y 361.393,Z 782.19,A -85,B 0,C 180,E1 9553.292,E2 9553.292} C_VEL
LIN {X 0,Y 365.893,Z 756.944,A -85,B 0,C 180,E1 9552.841,E2 9552.841} C_VEL
LIN {X 0,Y 372.896,Z 692.428,A -85,B 0,C 180,E1 9551.89,E2 9551.89} C_VEL
LIN {X 0,Y 381.599,Z 609.491,A -85,B 0,C 180,E1 9550.705,E2 9550.705} C_VEL
LIN {X 0,Y 379.208,Z 604.17,A -85,B 0,C 180,E1 9548.262,E2 9548.262} C_VEL
LIN {X 0,Y 377.638,Z 600.79,A -85,B 0,C 180,E1 9546.232,E2 9546.232} C_VEL
LIN {X 0,Y 376.358,Z 597.797,A -85,B 0,C 180,E1 9543.961,E2 9543.961} C_VEL
LIN {X 0,Y 375.281,Z 594.141,A -85,B 0,C 180,E1 9538.779,E2 9538.779} C_VEL
LIN {X 0,Y 376.678,Z 598.457,A -85,B 0,C 180,E1 9532.986,E2 9532.986} C_VEL
LIN {X 0,Y 378.554,Z 602.702,A -85,B 0,C 180,E1 9530.114,E2 9530.114} C_VEL
LIN {X 0,Y 381.113,Z 608.247,A -85,B 0,C 180,E1 9527.345,E2 9527.345} C_VEL
LIN {X 0,Y 381.535,Z 609.478,A -85,B 0,C 180,E1 9526.925,E2 9526.925} C_VEL
LIN {X 0,Y 366.559,Z 750.12,A -85,B 0,C 180,E1 9524.897,E2 9524.897} C_VEL
LIN {X 0,Y 362.076,Z 776.243,A -85,B 0,C 180,E1 9524.421,E2 9524.421} C_VEL
LIN {X 0,Y 357.091,Z 797.517,A -85,B 0,C 180,E1 9523.919,E2 9523.919} C_VEL
LIN {X 0,Y 349.505,Z 823.05,A -85,B 0,C 180,E1 9523.129,E2 9523.129} C_VEL
LIN {X 0,Y 342.116,Z 843.429,A -85,B 0,C 180,E1 9522.323,E2 9522.323} C_VEL
LIN {X 0,Y 332.658,Z 865.794,A -85,B 0,C 180,E1 9521.229,E2 9521.229} C_VEL
LIN {X 0,Y 322.871,Z 885.538,A -85,B 0,C 180,E1 9520.035,E2 9520.035} C_VEL
LIN {X 0,Y 311.943,Z 905.196,A -85,B 0,C 180,E1 9518.591,E2 9518.591} C_VEL
LIN {X 0,Y 299.268,Z 925.185,A -85,B 0,C 180,E1 9516.752,E2 9516.752} C_VEL
LIN {X 0,Y 287.263,Z 942.283,A -85,B 0,C 180,E1 9514.823,E2 9514.823} C_VEL
LIN {X 0,Y 273.305,Z 960.174,A -85,B 0,C 180,E1 9512.296,E2 9512.296} C_VEL
LIN {X 0,Y 260.637,Z 975.009,A -85,B 0,C 180,E1 9509.675,E2 9509.675} C_VEL
LIN {X 0,Y 245.784,Z 991.007,A -85,B 0,C 180,E1 9506.089,E2 9506.089} C_VEL
LIN {X 0,Y 233.332,Z 1003.421,A -85,B 0,C 180,E1 9502.518,E2 9502.518} C_VEL
LIN {X 0,Y 219.868,Z 1016.119,A -85,B 0,C 180,E1 9497.84,E2 9497.84} C_VEL
LIN {X 0,Y 208.522,Z 1026.262,A -85,B 0,C 180,E1 9492.915,E2 9492.915} C_VEL
LIN {X 0,Y 197.867,Z 1035.711,A -85,B 0,C 180,E1 9486.967,E2 9486.967} C_VEL
LIN {X 0,Y 189.27,Z 1043.262,A -85,B 0,C 180,E1 9480.474,E2 9480.474} C_VEL
LIN {X 0,Y 182.91,Z 1049.349,A -85,B 0,C 180,E1 9473.519,E2 9473.519} C_VEL
LIN {X 0,Y 178.653,Z 1053.939,A -85,B 0,C 180,E1 9465.917,E2 9465.917} C_VEL
LIN {X 0,Y 176.791,Z 1056.596,A -85,B 0,C 180,E1 9459.44,E2 9459.44} C_VEL
LIN {X 0,Y 176.123,Z 1058.214,A -85,B 0,C 180,E1 9452.929,E2 9452.929} C_VEL
LIN {X 0,Y 176.035,Z 1058.795,A -85,B 0,C 180,E1 9446.744,E2 9446.744} C_VEL
LIN {X 0,Y 176.331,Z 1058.329,A -85,B 0,C 180,E1 9440.205,E2 9440.205} C_VEL
LIN {X 0,Y 177.593,Z 1056.675,A -85,B 0,C 180,E1 9433.313,E2 9433.313} C_VEL
LIN {X 0,Y 180.275,Z 1054.027,A -85,B 0,C 180,E1 9426.809,E2 9426.809} C_VEL
LIN {X 0,Y 186.029,Z 1049.161,A -85,B 0,C 180,E1 9418.936,E2 9418.936} C_VEL
LIN {X 0,Y 193.375,Z 1043.272,A -85,B 0,C 180,E1 9412.4,E2 9412.4} C_VEL
LIN {X 0,Y 203.277,Z 1035.636,A -85,B 0,C 180,E1 9406.088,E2 9406.088} C_VEL
LIN {X 0,Y 214.645,Z 1026.486,A -85,B 0,C 180,E1 9400.597,E2 9400.597} C_VEL
LIN {X 0,Y 227.22,Z 1016.119,A -85,B 0,C 180,E1 9395.822,E2 9395.822} C_VEL
LIN {X 0,Y 241.451,Z 1003.523,A -85,B 0,C 180,E1 9391.452,E2 9391.452} C_VEL
LIN {X 0,Y 254.884,Z 990.848,A -85,B 0,C 180,E1 9388.035,E2 9388.035} C_VEL
LIN {X 0,Y 270.391,Z 974.862,A -85,B 0,C 180,E1 9384.7,E2 9384.7} C_VEL
LIN {X 0,Y 283.197,Z 960.454,A -85,B 0,C 180,E1 9382.324,E2 9382.324} C_VEL
LIN {X 0,Y 298.649,Z 941.253,A -85,B 0,C 180,E1 9379.814,E2 9379.814} C_VEL
LIN {X 0,Y 310.788,Z 924.449,A -85,B 0,C 180,E1 9378.065,E2 9378.065} C_VEL
LIN {X 0,Y 324.399,Z 903.332,A -85,B 0,C 180,E1 9376.289,E2 9376.289} C_VEL
LIN {X 0,Y 334.748,Z 885.127,A -85,B 0,C 180,E1 9375.062,E2 9375.062} C_VEL
LIN {X 0,Y 345.54,Z 863.698,A -85,B 0,C 180,E1 9373.871,E2 9373.871} C_VEL
LIN {X 0,Y 354.46,Z 842.805,A -85,B 0,C 180,E1 9372.937,E2 9372.937} C_VEL
LIN {X 0,Y 362.564,Z 820.768,A -85,B 0,C 180,E1 9372.136,E2 9372.136} C_VEL
LIN {X 0,Y 369.728,Z 796.587,A -85,B 0,C 180,E1 9371.452,E2 9371.452} C_VEL
LIN {X 0,Y 374.94,Z 774.526,A -85,B 0,C 180,E1 9370.974,E2 9370.974} C_VEL
LIN {X 0,Y 379.313,Z 748.676,A -85,B 0,C 180,E1 9370.541,E2 9370.541} C_VEL
LIN {X 0,Y 393.485,Z 619.026,A -85,B 0,C 180,E1 9368.733,E2 9368.733} C_VEL
LIN {X 0,Y 391.572,Z 614.717,A -85,B 0,C 180,E1 9366.304,E2 9366.304} C_VEL
LIN {X 0,Y 390.278,Z 611.67,A -85,B 0,C 180,E1 9363.967,E2 9363.967} C_VEL
LIN {X 0,Y 389.302,Z 608.455,A -85,B 0,C 180,E1 9358.97,E2 9358.97} C_VEL
LIN {X 0,Y 390.571,Z 612.326,A -85,B 0,C 180,E1 9353.754,E2 9353.754} C_VEL
LIN {X 0,Y 392.321,Z 616.461,A -85,B 0,C 180,E1 9350.982,E2 9350.982} C_VEL
LIN {X 0,Y 393.531,Z 619.223,A -85,B 0,C 180,E1 9349.54,E2 9349.54} C_VEL
LIN {X 0,Y 388.977,Z 661.307,A -85,B 0,C 180,E1 9348.962,E2 9348.962} C_VEL
LIN {X 0,Y 387.973,Z 669,A -85,B 0,C 180,E1 9348.997,E2 9348.997} C_VEL
LIN {X 0,Y 384.67,Z 689.553,A -85,B 0,C 180,E1 9349.629,E2 9349.629} C_VEL
LIN {X 0,Y 383.818,Z 696.159,A -85,B 0,C 180,E1 9349.655,E2 9349.655} C_VEL
LIN {X 0,Y 376.904,Z 756.796,A -85,B 0,C 180,E1 9348.812,E2 9348.812} C_VEL
LIN {X 0,Y 372.25,Z 781.89,A -85,B 0,C 180,E1 9348.402,E2 9348.402} C_VEL
LIN {X 0,Y 366.704,Z 804.231,A -85,B 0,C 180,E1 9347.969,E2 9347.969} C_VEL
LIN {X 0,Y 358.963,Z 828.627,A -85,B 0,C 180,E1 9347.357,E2 9347.357} C_VEL
LIN {X 0,Y 350.866,Z 849.8,A -85,B 0,C 180,E1 9346.669,E2 9346.669} C_VEL
LIN {X 0,Y 340.039,Z 873.702,A -85,B 0,C 180,E1 9345.673,E2 9345.673} C_VEL
LIN {X 0,Y 330.19,Z 892.523,A -85,B 0,C 180,E1 9344.685,E2 9344.685} C_VEL
LIN {X 0,Y 317.376,Z 914.095,A -85,B 0,C 180,E1 9343.285,E2 9343.285} C_VEL
LIN {X 0,Y 305.206,Z 932.124,A -85,B 0,C 180,E1 9341.819,E2 9341.819} C_VEL
LIN {X 0,Y 291.25,Z 950.871,A -85,B 0,C 180,E1 9339.921,E2 9339.921} C_VEL
LIN {X 0,Y 276.698,Z 968.201,A -85,B 0,C 180,E1 9337.683,E2 9337.683} C_VEL
LIN {X 0,Y 261.536,Z 984.812,A -85,B 0,C 180,E1 9334.97,E2 9334.97} C_VEL
LIN {X 0,Y 247.027,Z 999.13,A -85,B 0,C 180,E1 9331.933,E2 9331.933} C_VEL
LIN {X 0,Y 233.313,Z 1011.802,A -85,B 0,C 180,E1 9328.522,E2 9328.522} C_VEL
LIN {X 0,Y 217.945,Z 1024.975,A -85,B 0,C 180,E1 9323.848,E2 9323.848} C_VEL
LIN {X 0,Y 205.322,Z 1035.258,A -85,B 0,C 180,E1 9319.011,E2 9319.011} C_VEL
LIN {X 0,Y 192.83,Z 1045.07,A -85,B 0,C 180,E1 9312.787,E2 9312.787} C_VEL
LIN {X 0,Y 183.834,Z 1052.112,A -85,B 0,C 180,E1 9306.748,E2 9306.748} C_VEL
LIN {X 0,Y 175.756,Z 1058.78,A -85,B 0,C 180,E1 9298.919,E2 9298.919} C_VEL
LIN {X 0,Y 171.104,Z 1063.061,A -85,B 0,C 180,E1 9291.602,E2 9291.602} C_VEL
LIN {X 0,Y 168.662,Z 1066.053,A -85,B 0,C 180,E1 9284.067,E2 9284.067} C_VEL
LIN {X 0,Y 167.99,Z 1067.661,A -85,B 0,C 180,E1 9276.278,E2 9276.278} C_VEL
LIN {X 0,Y 168.04,Z 1067.91,A -85,B 0,C 180,E1 9270.341,E2 9270.341} C_VEL
LIN {X 0,Y 167.997,Z 1067.312,A -85,B 0,C 180,E1 9264.536,E2 9264.536} C_VEL
LIN {X 0,Y 168.321,Z 1065.647,A -85,B 0,C 180,E1 9258,E2 9258} C_VEL
LIN {X 0,Y 169.932,Z 1062.799,A -85,B 0,C 180,E1 9251.118,E2 9251.118} C_VEL
LIN {X 0,Y 174.136,Z 1057.897,A -85,B 0,C 180,E1 9243.024,E2 9243.024} C_VEL
LIN {X 0,Y 180.378,Z 1051.766,A -85,B 0,C 180,E1 9235.953,E2 9235.953} C_VEL
LIN {X 0,Y 189.469,Z 1043.746,A -85,B 0,C 180,E1 9228.996,E2 9228.996} C_VEL
LIN {X 0,Y 200.527,Z 1034.032,A -85,B 0,C 180,E1 9222.863,E2 9222.863} C_VEL
LIN {X 0,Y 212.499,Z 1023.486,A -85,B 0,C 180,E1 9217.767,E2 9217.767} C_VEL
LIN {X 0,Y 226.584,Z 1010.43,A -85,B 0,C 180,E1 9213.024,E2 9213.024} C_VEL
LIN {X 0,Y 239.836,Z 997.465,A -85,B 0,C 180,E1 9209.386,E2 9209.386} C_VEL
LIN {X 0,Y 254.701,Z 981.759,A -85,B 0,C 180,E1 9205.974,E2 9205.974} C_VEL
LIN {X 0,Y 267.18,Z 967.466,A -85,B 0,C 180,E1 9203.526,E2 9203.526} C_VEL
LIN {X 0,Y 281.346,Z 949.872,A -85,B 0,C 180,E1 9201.107,E2 9201.107} C_VEL
LIN {X 0,Y 294.267,Z 931.897,A -85,B 0,C 180,E1 9199.159,E2 9199.159} C_VEL
LIN {X 0,Y 306.661,Z 912.958,A -85,B 0,C 180,E1 9197.5,E2 9197.5} C_VEL
LIN {X 0,Y 318.42,Z 892.494,A -85,B 0,C 180,E1 9196.077,E2 9196.077} C_VEL
LIN {X 0,Y 328.138,Z 873.454,A -85,B 0,C 180,E1 9194.995,E2 9194.995} C_VEL
LIN {X 0,Y 338.437,Z 850.181,A -85,B 0,C 180,E1 9193.944,E2 9193.944} C_VEL
LIN {X 0,Y 346.136,Z 829.7,A -85,B 0,C 180,E1 9193.221,E2 9193.221} C_VEL
LIN {X 0,Y 353.642,Z 805.915,A -85,B 0,C 180,E1 9192.559,E2 9192.559} C_VEL
LIN {X 0,Y 359.282,Z 782.951,A -85,B 0,C 180,E1 9192.071,E2 9192.071} C_VEL
LIN {X 0,Y 363.861,Z 758.248,A -85,B 0,C 180,E1 9191.637,E2 9191.637} C_VEL
LIN {X 0,Y 369.823,Z 705.079,A -85,B 0,C 180,E1 9190.864,E2 9190.864} C_VEL
LIN {X 0,Y 379.411,Z 615.126,A -85,B 0,C 180,E1 9189.592,E2 9189.592} C_VEL
LIN {X 0,Y 376.924,Z 609.355,A -85,B 0,C 180,E1 9186.626,E2 9186.626} C_VEL
LIN {X 0,Y 375.23,Z 605.577,A -85,B 0,C 180,E1 9183.667,E2 9183.667} C_VEL
LIN {X 0,Y 374.3,Z 602.133,A -85,B 0,C 180,E1 9178.775,E2 9178.775} C_VEL
LIN {X 0,Y 375.612,Z 606.381,A -85,B 0,C 180,E1 9173.12,E2 9173.12} C_VEL
LIN {X 0,Y 377.382,Z 610.539,A -85,B 0,C 180,E1 9170.314,E2 9170.314} C_VEL
LIN {X 0,Y 379.368,Z 615.06,A -85,B 0,C 180,E1 9168.032,E2 9168.032} C_VEL
LIN {X 0,Y 364.694,Z 750.368,A -85,B 0,C 180,E1 9166.116,E2 9166.116} C_VEL
LIN {X 0,Y 360.131,Z 776.544,A -85,B 0,C 180,E1 9165.652,E2 9165.652} C_VEL
LIN {X 0,Y 355.077,Z 797.804,A -85,B 0,C 180,E1 9165.166,E2 9165.166} C_VEL
LIN {X 0,Y 347.273,Z 823.638,A -85,B 0,C 180,E1 9164.389,E2 9164.389} C_VEL
LIN {X 0,Y 339.775,Z 843.972,A -85,B 0,C 180,E1 9163.608,E2 9163.608} C_VEL
LIN {X 0,Y 329.731,Z 867.163,A -85,B 0,C 180,E1 9162.497,E2 9162.497} C_VEL
LIN {X 0,Y 319.79,Z 886.793,A -85,B 0,C 180,E1 9161.332,E2 9161.332} C_VEL
LIN {X 0,Y 308.34,Z 906.91,A -85,B 0,C 180,E1 9159.877,E2 9159.877} C_VEL
LIN {X 0,Y 295.765,Z 926.18,A -85,B 0,C 180,E1 9158.125,E2 9158.125} C_VEL
LIN {X 0,Y 282.715,Z 944.307,A -85,B 0,C 180,E1 9156.099,E2 9156.099} C_VEL
LIN {X 0,Y 268.855,Z 961.441,A -85,B 0,C 180,E1 9153.675,E2 9153.675} C_VEL
LIN {X 0,Y 255.887,Z 976.185,A -85,B 0,C 180,E1 9151.079,E2 9151.079} C_VEL
LIN {X 0,Y 240.634,Z 992.018,A -85,B 0,C 180,E1 9147.513,E2 9147.513} C_VEL
LIN {X 0,Y 228.091,Z 1004.089,A -85,B 0,C 180,E1 9144.025,E2 9144.025} C_VEL
LIN {X 0,Y 213.113,Z 1017.571,A -85,B 0,C 180,E1 9138.939,E2 9138.939} C_VEL
LIN {X 0,Y 201.571,Z 1027.448,A -85,B 0,C 180,E1 9133.985,E2 9133.985} C_VEL
LIN {X 0,Y 189.668,Z 1037.363,A -85,B 0,C 180,E1 9127.319,E2 9127.319} C_VEL
LIN {X 0,Y 181.615,Z 1044.116,A -85,B 0,C 180,E1 9121.166,E2 9121.166} C_VEL
LIN {X 0,Y 174.556,Z 1050.463,A -85,B 0,C 180,E1 9113.281,E2 9113.281} C_VEL
LIN {X 0,Y 170.625,Z 1054.488,A -85,B 0,C 180,E1 9105.987,E2 9105.987} C_VEL
LIN {X 0,Y 168.685,Z 1057.157,A -85,B 0,C 180,E1 9098.865,E2 9098.865} C_VEL
LIN {X 0,Y 168.089,Z 1058.673,A -85,B 0,C 180,E1 9091.704,E2 9091.704} C_VEL
LIN {X 0,Y 168.062,Z 1058.969,A -85,B 0,C 180,E1 9085.222,E2 9085.222} C_VEL
LIN {X 0,Y 168.488,Z 1058.341,A -85,B 0,C 180,E1 9078.706,E2 9078.706} C_VEL
LIN {X 0,Y 170.016,Z 1056.657,A -85,B 0,C 180,E1 9071.838,E2 9071.838} C_VEL
LIN {X 0,Y 173.784,Z 1053.449,A -85,B 0,C 180,E1 9064.07,E2 9064.07} C_VEL
LIN {X 0,Y 180.307,Z 1048.325,A -85,B 0,C 180,E1 9056.287,E2 9056.287} C_VEL
LIN {X 0,Y 188.55,Z 1042.257,A -85,B 0,C 180,E1 9049.686,E2 9049.686} C_VEL
LIN {X 0,Y 199.935,Z 1033.803,A -85,B 0,C 180,E1 9043.1,E2 9043.1} C_VEL
LIN {X 0,Y 211.107,Z 1025.277,A -85,B 0,C 180,E1 9038.164,E2 9038.164} C_VEL
LIN {X 0,Y 226.243,Z 1013.097,A -85,B 0,C 180,E1 9032.89,E2 9032.89} C_VEL
LIN {X 0,Y 239.37,Z 1001.756,A -85,B 0,C 180,E1 9029.187,E2 9029.187} C_VEL
LIN {X 0,Y 254.891,Z 987.33,A -85,B 0,C 180,E1 9025.545,E2 9025.545} C_VEL
LIN {X 0,Y 268.899,Z 972.996,A -85,B 0,C 180,E1 9022.751,E2 9022.751} C_VEL
LIN {X 0,Y 283.645,Z 956.609,A -85,B 0,C 180,E1 9020.21,E2 9020.21} C_VEL
LIN {X 0,Y 297.668,Z 939.089,A -85,B 0,C 180,E1 9018.081,E2 9018.081} C_VEL
LIN {X 0,Y 311.384,Z 920.222,A -85,B 0,C 180,E1 9016.235,E2 9016.235} C_VEL
LIN {X 0,Y 324.048,Z 900.26,A -85,B 0,C 180,E1 9014.683,E2 9014.683} C_VEL
LIN {X 0,Y 335.603,Z 879.878,A -85,B 0,C 180,E1 9013.402,E2 9013.402} C_VEL
LIN {X 0,Y 346.213,Z 857.957,A -85,B 0,C 180,E1 9012.294,E2 9012.294} C_VEL
LIN {X 0,Y 354.722,Z 837.758,A -85,B 0,C 180,E1 9011.47,E2 9011.47} C_VEL
LIN {X 0,Y 363.018,Z 814.145,A -85,B 0,C 180,E1 9010.697,E2 9010.697} C_VEL
LIN {X 0,Y 369.13,Z 792.82,A -85,B 0,C 180,E1 9010.141,E2 9010.141} C_VEL
LIN {X 0,Y 375.012,Z 766.175,A -85,B 0,C 180,E1 9009.618,E2 9009.618} C_VEL
LIN {X 0,Y 378.442,Z 743.895,A -85,B 0,C 180,E1 9009.279,E2 9009.279} C_VEL
LIN {X 0,Y 391.526,Z 625.127,A -85,B 0,C 180,E1 9007.631,E2 9007.631} C_VEL
LIN {X 0,Y 390.292,Z 622.227,A -85,B 0,C 180,E1 9005.882,E2 9005.882} C_VEL
LIN {X 0,Y 389.23,Z 619.551,A -85,B 0,C 180,E1 9003.83,E2 9003.83} C_VEL
LIN {X 0,Y 388.32,Z 616.451,A -85,B 0,C 180,E1 8998.967,E2 8998.967} C_VEL
LIN {X 0,Y 389.479,Z 620.134,A -85,B 0,C 180,E1 8993.958,E2 8993.958} C_VEL
LIN {X 0,Y 391.107,Z 624.154,A -85,B 0,C 180,E1 8991.25,E2 8991.25} C_VEL
LIN {X 0,Y 391.577,Z 625.466,A -85,B 0,C 180,E1 8990.612,E2 8990.612} C_VEL
LIN {X 0,Y 383.818,Z 696.159,A -85,B 0,C 180,E1 8989.655,E2 8989.655} C_VEL
LIN {X 0,Y 382.806,Z 703.857,A -85,B 0,C 180,E1 8989.703,E2 8989.703} C_VEL
LIN {X 0,Y 379.554,Z 724.404,A -85,B 0,C 180,E1 8990.352,E2 8990.352} C_VEL
LIN {X 0,Y 378.712,Z 731.006,A -85,B 0,C 180,E1 8990.373,E2 8990.373} C_VEL
LIN {X 0,Y 374.403,Z 763.566,A -85,B 0,C 180,E1 8989.913,E2 8989.913} C_VEL
LIN {X 0,Y 369.936,Z 785.777,A -85,B 0,C 180,E1 8989.553,E2 8989.553} C_VEL
LIN {X 0,Y 363.081,Z 811.326,A -85,B 0,C 180,E1 8989.046,E2 8989.046} C_VEL
LIN {X 0,Y 356.554,Z 830.814,A -85,B 0,C 180,E1 8988.553,E2 8988.553} C_VEL
LIN {X 0,Y 347.767,Z 853.173,A -85,B 0,C 180,E1 8987.839,E2 8987.839} C_VEL
LIN {X 0,Y 337.22,Z 875.538,A -85,B 0,C 180,E1 8986.915,E2 8986.915} C_VEL
LIN {X 0,Y 326.794,Z 894.969,A -85,B 0,C 180,E1 8985.912,E2 8985.912} C_VEL
LIN {X 0,Y 313.803,Z 916.07,A -85,B 0,C 180,E1 8984.553,E2 8984.553} C_VEL
LIN {X 0,Y 301.891,Z 933.296,A -85,B 0,C 180,E1 8983.175,E2 8983.175} C_VEL
LIN {X 0,Y 286.342,Z 953.416,A -85,B 0,C 180,E1 8981.141,E2 8981.141} C_VEL
LIN {X 0,Y 272.86,Z 969.042,A -85,B 0,C 180,E1 8979.138,E2 8979.138} C_VEL
LIN {X 0,Y 257.362,Z 985.48,A -85,B 0,C 180,E1 8976.476,E2 8976.476} C_VEL
LIN {X 0,Y 242.492,Z 999.713,A -85,B 0,C 180,E1 8973.48,E2 8973.48} C_VEL
LIN {X 0,Y 226.954,Z 1013.579,A -85,B 0,C 180,E1 8969.714,E2 8969.714} C_VEL
LIN {X 0,Y 211.85,Z 1025.867,A -85,B 0,C 180,E1 8965.21,E2 8965.21} C_VEL
LIN {X 0,Y 198.226,Z 1036.496,A -85,B 0,C 180,E1 8960.06,E2 8960.06} C_VEL
LIN {X 0,Y 185.84,Z 1045.617,A -85,B 0,C 180,E1 8953.953,E2 8953.953} C_VEL
LIN {X 0,Y 175.868,Z 1053.025,A -85,B 0,C 180,E1 8947.253,E2 8947.253} C_VEL
LIN {X 0,Y 167.748,Z 1059.227,A -85,B 0,C 180,E1 8939.26,E2 8939.26} C_VEL
LIN {X 0,Y 163.166,Z 1063.196,A -85,B 0,C 180,E1 8931.951,E2 8931.951} C_VEL
LIN {X 0,Y 160.515,Z 1066.259,A -85,B 0,C 180,E1 8923.326,E2 8923.326} C_VEL
LIN {X 0,Y 159.993,Z 1067.511,A -85,B 0,C 180,E1 8915.739,E2 8915.739} C_VEL
LIN {X 0,Y 160.051,Z 1067.671,A -85,B 0,C 180,E1 8910,E2 8910} C_VEL
LIN {X 0,Y 159.998,Z 1067.089,A -85,B 0,C 180,E1 8904.261,E2 8904.261} C_VEL
LIN {X 0,Y 160.393,Z 1065.414,A -85,B 0,C 180,E1 8897.397,E2 8897.397} C_VEL
LIN {X 0,Y 162.21,Z 1062.558,A -85,B 0,C 180,E1 8890.182,E2 8890.182} C_VEL
LIN {X 0,Y 167.087,Z 1057.38,A -85,B 0,C 180,E1 8881.397,E2 8881.397} C_VEL
LIN {X 0,Y 173.95,Z 1051.191,A -85,B 0,C 180,E1 8874.104,E2 8874.104} C_VEL
LIN {X 0,Y 184.077,Z 1042.81,A -85,B 0,C 180,E1 8866.81,E2 8866.81} C_VEL
LIN {X 0,Y 195.529,Z 1033.277,A -85,B 0,C 180,E1 8860.814,E2 8860.814} C_VEL
LIN {X 0,Y 208.793,Z 1022.136,A -85,B 0,C 180,E1 8855.5,E2 8855.5} C_VEL
LIN {X 0,Y 222.871,Z 1009.473,A -85,B 0,C 180,E1 8851.029,E2 8851.029} C_VEL
LIN {X 0,Y 237.376,Z 995.722,A -85,B 0,C 180,E1 8847.279,E2 8847.279} C_VEL
LIN {X 0,Y 251.975,Z 980.561,A -85,B 0,C 180,E1 8844.121,E2 8844.121} C_VEL
LIN {X 0,Y 265.626,Z 965.239,A -85,B 0,C 180,E1 8841.6,E2 8841.6} C_VEL
LIN {X 0,Y 281.011,Z 946.124,A -85,B 0,C 180,E1 8839.144,E2 8839.144} C_VEL
LIN {X 0,Y 293.403,Z 929.045,A -85,B 0,C 180,E1 8837.405,E2 8837.405} C_VEL
LIN {X 0,Y 307.394,Z 907.422,A -85,B 0,C 180,E1 8835.663,E2 8835.663} C_VEL
LIN {X 0,Y 318.047,Z 888.773,A -85,B 0,C 180,E1 8834.465,E2 8834.465} C_VEL
LIN {X 0,Y 329.303,Z 866.351,A -85,B 0,C 180,E1 8833.305,E2 8833.305} C_VEL
LIN {X 0,Y 338.031,Z 846.016,A -85,B 0,C 180,E1 8832.47,E2 8832.47} C_VEL
LIN {X 0,Y 346.679,Z 822.568,A -85,B 0,C 180,E1 8831.711,E2 8831.711} C_VEL
LIN {X 0,Y 353.619,Z 798.987,A -85,B 0,C 180,E1 8831.136,E2 8831.136} C_VEL
LIN {X 0,Y 359.328,Z 774.575,A -85,B 0,C 180,E1 8830.669,E2 8830.669} C_VEL
LIN {X 0,Y 363.205,Z 750.195,A -85,B 0,C 180,E1 8830.28,E2 8830.28} C_VEL
LIN {X 0,Y 377.338,Z 620.996,A -85,B 0,C 180,E1 8828.465,E2 8828.465} C_VEL
LIN {X 0,Y 375.456,Z 616.572,A -85,B 0,C 180,E1 8825.962,E2 8825.962} C_VEL
LIN {X 0,Y 374.181,Z 613.455,A -85,B 0,C 180,E1 8823.524,E2 8823.524} C_VEL
LIN {X 0,Y 373.307,Z 610.23,A -85,B 0,C 180,E1 8818.619,E2 8818.619} C_VEL
LIN {X 0,Y 374.514,Z 614.191,A -85,B 0,C 180,E1 8813.331,E2 8813.331} C_VEL
LIN {X 0,Y 376.161,Z 618.235,A -85,B 0,C 180,E1 8810.591,E2 8810.591} C_VEL
LIN {X 0,Y 377.304,Z 621.025,A -85,B 0,C 180,E1 8809.145,E2 8809.145} C_VEL
LIN {X 0,Y 362.994,Z 750.615,A -85,B 0,C 180,E1 8807.347,E2 8807.347} C_VEL
LIN {X 0,Y 358.383,Z 776.712,A -85,B 0,C 180,E1 8806.899,E2 8806.899} C_VEL
LIN {X 0,Y 353.225,Z 798.122,A -85,B 0,C 180,E1 8806.426,E2 8806.426} C_VEL
LIN {X 0,Y 345.659,Z 822.949,A -85,B 0,C 180,E1 8805.709,E2 8805.709} C_VEL
LIN {X 0,Y 338.053,Z 843.393,A -85,B 0,C 180,E1 8804.954,E2 8804.954} C_VEL
LIN {X 0,Y 328.741,Z 864.964,A -85,B 0,C 180,E1 8803.974,E2 8803.974} C_VEL
LIN {X 0,Y 318.186,Z 885.639,A -85,B 0,C 180,E1 8802.806,E2 8802.806} C_VEL
LIN {X 0,Y 306.908,Z 905.258,A -85,B 0,C 180,E1 8801.453,E2 8801.453} C_VEL
LIN {X 0,Y 293.697,Z 925.372,A -85,B 0,C 180,E1 8799.708,E2 8799.708} C_VEL
LIN {X 0,Y 281.589,Z 941.945,A -85,B 0,C 180,E1 8797.938,E2 8797.938} C_VEL
LIN {X 0,Y 266.157,Z 960.88,A -85,B 0,C 180,E1 8795.386,E2 8795.386} C_VEL
LIN {X 0,Y 252.825,Z 975.694,A -85,B 0,C 180,E1 8792.854,E2 8792.854} C_VEL
LIN {X 0,Y 236.713,Z 992.009,A -85,B 0,C 180,E1 8789.262,E2 8789.262} C_VEL
LIN {X 0,Y 223.669,Z 1004.158,A -85,B 0,C 180,E1 8785.794,E2 8785.794} C_VEL
LIN {X 0,Y 208.646,Z 1017.213,A -85,B 0,C 180,E1 8780.927,E2 8780.927} C_VEL
LIN {X 0,Y 196.884,Z 1026.835,A -85,B 0,C 180,E1 8776.15,E2 8776.15} C_VEL
LIN {X 0,Y 185.094,Z 1036.253,A -85,B 0,C 180,E1 8770.004,E2 8770.004} C_VEL
LIN {X 0,Y 175.429,Z 1043.788,A -85,B 0,C 180,E1 8763.173,E2 8763.173} C_VEL
LIN {X 0,Y 167.887,Z 1050.102,A -85,B 0,C 180,E1 8755.392,E2 8755.392} C_VEL
LIN {X 0,Y 163.02,Z 1054.573,A -85,B 0,C 180,E1 8747.122,E2 8747.122} C_VEL
LIN {X 0,Y 160.88,Z 1057.168,A -85,B 0,C 180,E1 8740.022,E2 8740.022} C_VEL
LIN {X 0,Y 160.109,Z 1058.838,A -85,B 0,C 180,E1 8732.267,E2 8732.267} C_VEL
LIN {X 0,Y 160.056,Z 1059.223,A -85,B 0,C 180,E1 8725.701,E2 8725.701} C_VEL
LIN {X 0,Y 160.511,Z 1058.611,A -85,B 0,C 180,E1 8718.501,E2 8718.501} C_VEL
LIN {X 0,Y 162.153,Z 1056.967,A -85,B 0,C 180,E1 8711.298,E2 8711.298} C_VEL
LIN {X 0,Y 165.963,Z 1053.953,A -85,B 0,C 180,E1 8703.523,E2 8703.523} C_VEL
LIN {X 0,Y 173.154,Z 1048.748,A -85,B 0,C 180,E1 8695.084,E2 8695.084} C_VEL
LIN {X 0,Y 181.86,Z 1042.73,A -85,B 0,C 180,E1 8688.297,E2 8688.297} C_VEL
LIN {X 0,Y 194.363,Z 1033.962,A -85,B 0,C 180,E1 8681.315,E2 8681.315} C_VEL
LIN {X 0,Y 206.413,Z 1025.189,A -85,B 0,C 180,E1 8676.227,E2 8676.227} C_VEL
LIN {X 0,Y 221.852,Z 1013.231,A -85,B 0,C 180,E1 8671.093,E2 8671.093} C_VEL
LIN {X 0,Y 235.447,Z 1001.881,A -85,B 0,C 180,E1 8667.43,E2 8667.43} C_VEL
LIN {X 0,Y 251.444,Z 987.434,A -85,B 0,C 180,E1 8663.849,E2 8663.849} C_VEL
LIN {X 0,Y 265.821,Z 973.094,A -85,B 0,C 180,E1 8661.115,E2 8661.115} C_VEL
LIN {X 0,Y 281.159,Z 956.384,A -85,B 0,C 180,E1 8658.602,E2 8658.602} C_VEL
LIN {X 0,Y 294.798,Z 939.696,A -85,B 0,C 180,E1 8656.629,E2 8656.629} C_VEL
LIN {X 0,Y 308.318,Z 921.484,A -85,B 0,C 180,E1 8654.888,E2 8654.888} C_VEL
LIN {X 0,Y 321.185,Z 901.731,A -85,B 0,C 180,E1 8653.381,E2 8653.381} C_VEL
LIN {X 0,Y 331.998,Z 883.105,A -85,B 0,C 180,E1 8652.229,E2 8652.229} C_VEL
LIN {X 0,Y 343.585,Z 860.065,A -85,B 0,C 180,E1 8651.074,E2 8651.074} C_VEL
LIN {X 0,Y 352.069,Z 840.421,A -85,B 0,C 180,E1 8650.285,E2 8650.285} C_VEL
LIN {X 0,Y 360.677,Z 816.899,A -85,B 0,C 180,E1 8649.52,E2 8649.52} C_VEL
LIN {X 0,Y 367.215,Z 794.695,A -85,B 0,C 180,E1 8648.953,E2 8648.953} C_VEL
LIN {X 0,Y 372.937,Z 770.193,A -85,B 0,C 180,E1 8648.473,E2 8648.473} C_VEL
LIN {X 0,Y 376.783,Z 746.415,A -85,B 0,C 180,E1 8648.115,E2 8648.115} C_VEL
LIN {X 0,Y 389.739,Z 631.344,A -85,B 0,C 180,E1 8646.563,E2 8646.563} C_VEL
LIN {X 0,Y 388.184,Z 627.432,A -85,B 0,C 180,E1 8643.692,E2 8643.692} C_VEL
LIN {X 0,Y 387.351,Z 624.331,A -85,B 0,C 180,E1 8639.113,E2 8639.113} C_VEL
LIN {X 0,Y 388.422,Z 628.053,A -85,B 0,C 180,E1 8634.09,E2 8634.09} C_VEL
LIN {X 0,Y 389.773,Z 631.614,A -85,B 0,C 180,E1 8631.694,E2 8631.694} C_VEL
LIN {X 0,Y 378.712,Z 731.006,A -85,B 0,C 180,E1 8630.373,E2 8630.373} C_VEL
LIN {X 0,Y 377.714,Z 738.699,A -85,B 0,C 180,E1 8630.42,E2 8630.42} C_VEL
LIN {X 0,Y 374.069,Z 759.173,A -85,B 0,C 180,E1 8631.091,E2 8631.091} C_VEL
LIN {X 0,Y 372.793,Z 765.718,A -85,B 0,C 180,E1 8631.095,E2 8631.095} C_VEL
LIN {X 0,Y 367.835,Z 789.395,A -85,B 0,C 180,E1 8630.721,E2 8630.721} C_VEL
LIN {X 0,Y 361.168,Z 813.019,A -85,B 0,C 180,E1 8630.259,E2 8630.259} C_VEL
LIN {X 0,Y 354.164,Z 833.38,A -85,B 0,C 180,E1 8629.755,E2 8629.755} C_VEL
LIN {X 0,Y 344.297,Z 857.319,A -85,B 0,C 180,E1 8628.992,E2 8628.992} C_VEL
LIN {X 0,Y 334.562,Z 877.375,A -85,B 0,C 180,E1 8628.176,E2 8628.176} C_VEL
